KUKA KRL program: EPS_2_25999_MH4A_A_20251114084358.src

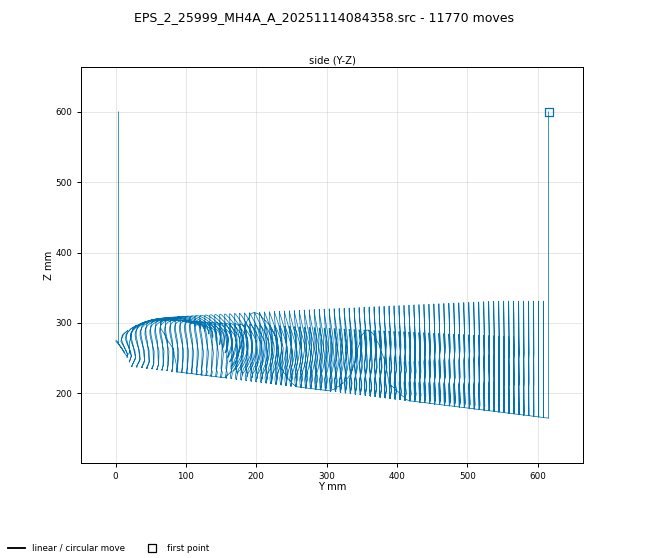
[picture p0: tool path of EPS_2_25999_MH4A_A_20251114084358.src, 11770 of 11772 moves have a stored position in this frame; points joined in program order, loops and branches not executed]
&ACCESS RVP
&REL 4
&COMMENT QRS 19112012
&PARAM EDITMASK = *
DEF PART()
EXT BAS (BAS_COMMAND :IN,REAL :IN )
INT I
BAS (#INITMOV,0 )

;KUKA QRS Post kuka4.cps  Date:22-06-2017 !

File_ID=2914

QRS_PRE_INIT()

;Init var - Until changes are made in qrs_pre_init
Outlet_Square_prg=0
Inlet_1_Square_prg=0
Inlet_2_Square_prg=0
Inlet_3_Square_prg=0
Inlet_4_Square_prg=0
Inlet_5_Square_prg=0

Outlet_1={X 0.000, Y 541.800, Z 256.000, B 0.000, E1 0.000 }
Inlet_1={X 0.000, Y 548.610, Z 213.500, B 0.000, E1 225.000 }
Outlet_1_type=150
Inlet_1_type=135
;QRS#1=Sidecore dimensions
;QRS#2=150-6" PVC SDR 28
;QRS#3=135-5" PVC SDR 28
;QRS#4=
;QRS#5=
;QRS#6=
;QRS#7=
;QRS#8=
;QRS#9=10-06 PSX
;QRS#10=8-11 PSX
;QRS#11=
;QRS#12=
;QRS#13=
;QRS#14=
;QRS#15=
;QRS#16=1220x127x610 2'
;QRS#17=EPS Height
;QRS#18=331
;QRS#19=*
;QRS#20= UPDATED VERSION 22-06-2017
;QRS#21=*
Outlet_Square=070
Inlet_1_Square=070
Inlet_2_Square=0
Inlet_3_Square=0
Inlet_4_Square=0
Inlet_5_Square=0
Mill_Square=1
Outlet_Square_Prg=203
Inlet_1_Square_prg=202

QRS_INIT()

$ADVANCE=5

; T1
PTP {E1 173.61,E2 173.61}
PTP {X 0,Y 615.503,A -85,B 0,C 180,E1 173.61,E2 173.61,E3 0,E4 0,E5 0,E6 0}
QRS_SPEED_INIT()
LIN {X 0,Y 615.503,Z 600,A -85,B 0,C 180,E1 173.61,E2 173.61,E3 0,E4 0,E5 0,E6 0} C_VEL
LIN {X 0,Y 615.503,Z 174.687,A -85,B 0,C 180,E1 173.61,E2 173.61} C_VEL
LIN {X 0,Y 615.503,Z 166.515,A -85,B 0,C 180,E1 173.61,E2 173.61} C_VEL
LIN {X 0,Y 615.489,Z 164.515,A -85,B 0,C 180,E1 173.424,E2 173.424} C_VEL
LIN {X 0,Y 615.497,Z 164.512,A -85,B 0,C 180,E1 170.802,E2 170.802} C_VEL
LIN {X 0,Y 615.481,Z 164.513,A -85,B 0,C 180,E1 168.14,E2 168.14} C_VEL
LIN {X 0,Y 615.485,Z 164.51,A -85,B 0,C 180,E1 165.452,E2 165.452} C_VEL
LIN {X 0,Y 615.477,Z 164.51,A -85,B 0,C 180,E1 162.73,E2 162.73} C_VEL
LIN {X 0,Y 615.462,Z 164.512,A -85,B 0,C 180,E1 159.967,E2 159.967} C_VEL
LIN {X 0,Y 615.491,Z 164.508,A -85,B 0,C 180,E1 157.156,E2 157.156} C_VEL
LIN {X 0,Y 615.498,Z 164.512,A -85,B 0,C 180,E1 154.286,E2 154.286} C_VEL
LIN {X 0,Y 615.493,Z 164.507,A -85,B 0,C 180,E1 151.343,E2 151.343} C_VEL
LIN {X 0,Y 615.477,Z 164.512,A -85,B 0,C 180,E1 148.916,E2 148.916} C_VEL
LIN {X 0,Y 615.487,Z 164.512,A -85,B 0,C 180,E1 146.466,E2 146.466} C_VEL
LIN {X 0,Y 615.49,Z 164.507,A -85,B 0,C 180,E1 143.577,E2 143.577} C_VEL
LIN {X 0,Y 615.463,Z 164.512,A -85,B 0,C 180,E1 140.941,E2 140.941} C_VEL
LIN {X 0,Y 615.467,Z 164.513,A -85,B 0,C 180,E1 138.526,E2 138.526} C_VEL
LIN {X 0,Y 615.494,Z 164.506,A -85,B 0,C 180,E1 135.852,E2 135.852} C_VEL
LIN {X 0,Y 615.463,Z 164.513,A -85,B 0,C 180,E1 133.046,E2 133.046} C_VEL
LIN {X 0,Y 615.46,Z 164.513,A -85,B 0,C 180,E1 130.609,E2 130.609} C_VEL
LIN {X 0,Y 615.488,Z 164.507,A -85,B 0,C 180,E1 128.014,E2 128.014} C_VEL
LIN {X 0,Y 615.474,Z 164.51,A -85,B 0,C 180,E1 125.617,E2 125.617} C_VEL
LIN {X 0,Y 615.468,Z 164.512,A -85,B 0,C 180,E1 123.238,E2 123.238} C_VEL
LIN {X 0,Y 615.485,Z 164.512,A -85,B 0,C 180,E1 120.92,E2 120.92} C_VEL
LIN {X 0,Y 615.496,Z 164.512,A -85,B 0,C 180,E1 118.454,E2 118.454} C_VEL
LIN {X 0,Y 615.468,Z 164.512,A -85,B 0,C 180,E1 115.567,E2 115.567} C_VEL
LIN {X 0,Y 615.476,Z 164.51,A -85,B 0,C 180,E1 112.845,E2 112.845} C_VEL
LIN {X 0,Y 615.481,Z 164.509,A -85,B 0,C 180,E1 110.033,E2 110.033} C_VEL
LIN {X 0,Y 615.471,Z 164.514,A -85,B 0,C 180,E1 107.271,E2 107.271} C_VEL
LIN {X 0,Y 615.494,Z 164.512,A -85,B 0,C 180,E1 104.549,E2 104.549} C_VEL
LIN {X 0,Y 615.486,Z 164.514,A -85,B 0,C 180,E1 101.861,E2 101.861} C_VEL
LIN {X 0,Y 615.494,Z 164.51,A -85,B 0,C 180,E1 99.199,E2 99.199} C_VEL
LIN {X 0,Y 615.477,Z 164.512,A -85,B 0,C 180,E1 96.557,E2 96.557} C_VEL
LIN {X 0,Y 615.472,Z 164.512,A -85,B 0,C 180,E1 93.929,E2 93.929} C_VEL
LIN {X 0,Y 615.488,Z 164.508,A -85,B 0,C 180,E1 91.309,E2 91.309} C_VEL
LIN {X 0,Y 615.474,Z 164.511,A -85,B 0,C 180,E1 88.692,E2 88.692} C_VEL
LIN {X 0,Y 615.464,Z 164.512,A -85,B 0,C 180,E1 86.071,E2 86.071} C_VEL
LIN {X 0,Y 615.487,Z 164.507,A -85,B 0,C 180,E1 83.412,E2 83.412} C_VEL
LIN {X 0,Y 615.475,Z 164.51,A -85,B 0,C 180,E1 80.801,E2 80.801} C_VEL
LIN {X 0,Y 615.464,Z 164.513,A -85,B 0,C 180,E1 78.139,E2 78.139} C_VEL
LIN {X 0,Y 615.476,Z 164.51,A -85,B 0,C 180,E1 76.799,E2 76.799} C_VEL
LIN {X 0,Y 615.481,Z 165.4,A -85,B 0,C 180,E1 76.065,E2 76.065} C_VEL
LIN {X 0,Y 615.489,Z 170.184,A -85,B 0,C 180,E1 73.413,E2 73.413} C_VEL
LIN {X 0,Y 615.478,Z 175.208,A -85,B 0,C 180,E1 70.662,E2 70.662} C_VEL
LIN {X 0,Y 615.453,Z 179.147,A -85,B 0,C 180,E1 68.567,E2 68.567} C_VEL
LIN {X 0,Y 615.485,Z 184.575,A -85,B 0,C 180,E1 65.728,E2 65.728} C_VEL
LIN {X 0,Y 615.43,Z 190.251,A -85,B 0,C 180,E1 62.82,E2 62.82} C_VEL
LIN {X 0,Y 615.497,Z 195.416,A -85,B 0,C 180,E1 60.202,E2 60.202} C_VEL
LIN {X 0,Y 615.471,Z 200.75,A -85,B 0,C 180,E1 57.542,E2 57.542} C_VEL
LIN {X 0,Y 615.477,Z 205.521,A -85,B 0,C 180,E1 55.184,E2 55.184} C_VEL
LIN {X 0,Y 615.486,Z 209.216,A -85,B 0,C 180,E1 53.367,E2 53.367} C_VEL
LIN {X 0,Y 615.484,Z 219.857,A -85,B 0,C 180,E1 53.062,E2 53.062} C_VEL
LIN {X 0,Y 615.474,Z 228.721,A -85,B 0,C 180,E1 52.709,E2 52.709} C_VEL
LIN {X 0,Y 615.482,Z 237.063,A -85,B 0,C 180,E1 52.276,E2 52.276} C_VEL
LIN {X 0,Y 615.489,Z 246.817,A -85,B 0,C 180,E1 51.619,E2 51.619} C_VEL
LIN {X 0,Y 615.496,Z 254.636,A -85,B 0,C 180,E1 50.935,E2 50.935} C_VEL
LIN {X 0,Y 615.499,Z 260.962,A -85,B 0,C 180,E1 50.251,E2 50.251} C_VEL
LIN {X 0,Y 615.495,Z 267.278,A -85,B 0,C 180,E1 49.394,E2 49.394} C_VEL
LIN {X 0,Y 615.495,Z 272.077,A -85,B 0,C 180,E1 48.527,E2 48.527} C_VEL
LIN {X 0,Y 615.496,Z 275.715,A -85,B 0,C 180,E1 47.648,E2 47.648} C_VEL
LIN {X 0,Y 615.495,Z 278.295,A -85,B 0,C 180,E1 46.756,E2 46.756} C_VEL
LIN {X 0,Y 615.492,Z 279.859,A -85,B 0,C 180,E1 45.851,E2 45.851} C_VEL
LIN {X 0,Y 615.498,Z 280.387,A -85,B 0,C 180,E1 44.932,E2 44.932} C_VEL
LIN {X 0,Y 615.493,Z 279.772,A -85,B 0,C 180,E1 43.998,E2 43.998} C_VEL
LIN {X 0,Y 615.493,Z 278.038,A -85,B 0,C 180,E1 43.048,E2 43.048} C_VEL
LIN {X 0,Y 615.499,Z 276.021,A -85,B 0,C 180,E1 42.351,E2 42.351} C_VEL
LIN {X 0,Y 615.493,Z 272.484,A -85,B 0,C 180,E1 41.472,E2 41.472} C_VEL
LIN {X 0,Y 615.494,Z 267.808,A -85,B 0,C 180,E1 40.605,E2 40.605} C_VEL
LIN {X 0,Y 615.497,Z 261.727,A -85,B 0,C 180,E1 39.748,E2 39.748} C_VEL
LIN {X 0,Y 615.496,Z 255.543,A -85,B 0,C 180,E1 39.063,E2 39.063} C_VEL
LIN {X 0,Y 615.491,Z 249.179,A -85,B 0,C 180,E1 38.484,E2 38.484} C_VEL
LIN {X 0,Y 615.445,Z 241.506,A -85,B 0,C 180,E1 37.912,E2 37.912} C_VEL
LIN {X 0,Y 615.443,Z 231.76,A -85,B 0,C 180,E1 37.339,E2 37.339} C_VEL
LIN {X 0,Y 615.473,Z 222.384,A -85,B 0,C 180,E1 36.935,E2 36.935} C_VEL
LIN {X 0,Y 615.497,Z 213.181,A -85,B 0,C 180,E1 36.646,E2 36.646} C_VEL
LIN {X 0,Y 615.488,Z 209.2,A -85,B 0,C 180,E1 36.535,E2 36.535} C_VEL
LIN {X 0,Y 615.462,Z 204.091,A -85,B 0,C 180,E1 34.023,E2 34.023} C_VEL
LIN {X 0,Y 615.48,Z 199.37,A -85,B 0,C 180,E1 31.685,E2 31.685} C_VEL
LIN {X 0,Y 615.482,Z 194.823,A -85,B 0,C 180,E1 29.406,E2 29.406} C_VEL
LIN {X 0,Y 615.474,Z 190.147,A -85,B 0,C 180,E1 27.042,E2 27.042} C_VEL
LIN {X 0,Y 615.486,Z 184.746,A -85,B 0,C 180,E1 24.271,E2 24.271} C_VEL
LIN {X 0,Y 615.446,Z 180.666,A -85,B 0,C 180,E1 22.137,E2 22.137} C_VEL
LIN {X 0,Y 615.428,Z 176.69,A -85,B 0,C 180,E1 20.034,E2 20.034} C_VEL
LIN {X 0,Y 615.495,Z 171.608,A -85,B 0,C 180,E1 17.27,E2 17.27} C_VEL
LIN {X 0,Y 615.465,Z 166.69,A -85,B 0,C 180,E1 14.549,E2 14.549} C_VEL
LIN {X 0,Y 615.496,Z 164.508,A -85,B 0,C 180,E1 13.2,E2 13.2} C_VEL
LIN {X 0,Y 615.474,Z 164.512,A -85,B 0,C 180,E1 10.526,E2 10.526} C_VEL
LIN {X 0,Y 615.487,Z 164.514,A -85,B 0,C 180,E1 7.875,E2 7.875} C_VEL
LIN {X 0,Y 615.491,Z 164.509,A -85,B 0,C 180,E1 5.241,E2 5.241} C_VEL
LIN {X 0,Y 615.47,Z 164.512,A -85,B 0,C 180,E1 2.617,E2 2.617} C_VEL
LIN {X 0,Y 615.482,Z 164.512,A -85,B 0,C 180,E1 -0.001,E2 -0.001} C_VEL
LIN {X 0,Y 615.489,Z 164.512,A -85,B 0,C 180,E1 -2.618,E2 -2.618} C_VEL
LIN {X 0,Y 615.471,Z 164.512,A -85,B 0,C 180,E1 -5.242,E2 -5.242} C_VEL
LIN {X 0,Y 615.474,Z 164.512,A -85,B 0,C 180,E1 -7.876,E2 -7.876} C_VEL
LIN {X 0,Y 615.493,Z 164.514,A -85,B 0,C 180,E1 -10.527,E2 -10.527} C_VEL
LIN {X 0,Y 615.473,Z 164.512,A -85,B 0,C 180,E1 -13.202,E2 -13.202} C_VEL
LIN {X 0,Y 615.489,Z 164.509,A -85,B 0,C 180,E1 -15.906,E2 -15.906} C_VEL
LIN {X 0,Y 615.49,Z 164.512,A -85,B 0,C 180,E1 -18.646,E2 -18.646} C_VEL
LIN {X 0,Y 615.475,Z 164.511,A -85,B 0,C 180,E1 -21.433,E2 -21.433} C_VEL
LIN {X 0,Y 615.489,Z 164.515,A -85,B 0,C 180,E1 -24.272,E2 -24.272} C_VEL
LIN {X 0,Y 615.469,Z 164.513,A -85,B 0,C 180,E1 -27.041,E2 -27.041} C_VEL
LIN {X 0,Y 615.497,Z 164.509,A -85,B 0,C 180,E1 -29.796,E2 -29.796} C_VEL
LIN {X 0,Y 615.482,Z 164.513,A -85,B 0,C 180,E1 -32.458,E2 -32.458} C_VEL
LIN {X 0,Y 615.485,Z 164.512,A -85,B 0,C 180,E1 -34.816,E2 -34.816} C_VEL
LIN {X 0,Y 615.493,Z 164.508,A -85,B 0,C 180,E1 -37.242,E2 -37.242} C_VEL
LIN {X 0,Y 615.483,Z 164.512,A -85,B 0,C 180,E1 -40.088,E2 -40.088} C_VEL
LIN {X 0,Y 615.478,Z 164.513,A -85,B 0,C 180,E1 -42.354,E2 -42.354} C_VEL
LIN {X 0,Y 615.494,Z 164.511,A -85,B 0,C 180,E1 -45.068,E2 -45.068} C_VEL
LIN {X 0,Y 615.472,Z 164.512,A -85,B 0,C 180,E1 -47.922,E2 -47.922} C_VEL
LIN {X 0,Y 615.469,Z 164.513,A -85,B 0,C 180,E1 -50.248,E2 -50.248} C_VEL
LIN {X 0,Y 615.492,Z 164.512,A -85,B 0,C 180,E1 -53.063,E2 -53.063} C_VEL
LIN {X 0,Y 615.472,Z 164.513,A -85,B 0,C 180,E1 -55.977,E2 -55.977} C_VEL
LIN {X 0,Y 615.474,Z 164.512,A -85,B 0,C 180,E1 -58.314,E2 -58.314} C_VEL
LIN {X 0,Y 615.478,Z 164.615,A -85,B 0,C 180,E1 -59.46,E2 -59.46} C_VEL
LIN {X 0,Y 615.479,Z 174.178,A -85,B 0,C 180,E1 -62.085,E2 -62.085} C_VEL
LIN {X 0,Y 615.463,Z 185.21,A -85,B 0,C 180,E1 -65.007,E2 -65.007} C_VEL
LIN {X 0,Y 615.452,Z 193.485,A -85,B 0,C 180,E1 -67.154,E2 -67.154} C_VEL
LIN {X 0,Y 615.469,Z 203.484,A -85,B 0,C 180,E1 -69.709,E2 -69.709} C_VEL
LIN {X 0,Y 615.495,Z 214.135,A -85,B 0,C 180,E1 -72.387,E2 -72.387} C_VEL
LIN {X 0,Y 615.473,Z 225.145,A -85,B 0,C 180,E1 -75.112,E2 -75.112} C_VEL
LIN {X 0,Y 615.479,Z 236.141,A -85,B 0,C 180,E1 -77.805,E2 -77.805} C_VEL
LIN {X 0,Y 615.489,Z 247.136,A -85,B 0,C 180,E1 -80.47,E2 -80.47} C_VEL
LIN {X 0,Y 615.485,Z 248.505,A -85,B 0,C 180,E1 -80.801,E2 -80.801} C_VEL
LIN {X 0,Y 615.495,Z 260.895,A -85,B 0,C 180,E1 -81.091,E2 -81.091} C_VEL
LIN {X 0,Y 615.471,Z 271.229,A -85,B 0,C 180,E1 -81.463,E2 -81.463} C_VEL
LIN {X 0,Y 615.474,Z 279.916,A -85,B 0,C 180,E1 -81.877,E2 -81.877} C_VEL
LIN {X 0,Y 615.492,Z 288.199,A -85,B 0,C 180,E1 -82.372,E2 -82.372} C_VEL
LIN {X 0,Y 615.499,Z 295.935,A -85,B 0,C 180,E1 -82.942,E2 -82.942} C_VEL
LIN {X 0,Y 615.498,Z 301.647,A -85,B 0,C 180,E1 -83.444,E2 -83.444} C_VEL
LIN {X 0,Y 615.5,Z 307.922,A -85,B 0,C 180,E1 -84.102,E2 -84.102} C_VEL
LIN {X 0,Y 615.495,Z 313.136,A -85,B 0,C 180,E1 -84.759,E2 -84.759} C_VEL
LIN {X 0,Y 615.495,Z 317.483,A -85,B 0,C 180,E1 -85.416,E2 -85.416} C_VEL
LIN {X 0,Y 615.491,Z 322.604,A -85,B 0,C 180,E1 -86.399,E2 -86.399} C_VEL
LIN {X 0,Y 615.488,Z 325.221,A -85,B 0,C 180,E1 -87.055,E2 -87.055} C_VEL
LIN {X 0,Y 615.499,Z 328.085,A -85,B 0,C 180,E1 -88.037,E2 -88.037} C_VEL
LIN {X 0,Y 615.493,Z 329.33,A -85,B 0,C 180,E1 -88.692,E2 -88.692} C_VEL
LIN {X 0,Y 615.491,Z 330.104,A -85,B 0,C 180,E1 -89.346,E2 -89.346} C_VEL
LIN {X 0,Y 615.491,Z 330.389,A -85,B 0,C 180,E1 -90,E2 -90} C_VEL
LIN {X 0,Y 615.491,Z 330.104,A -85,B 0,C 180,E1 -90.654,E2 -90.654} C_VEL
LIN {X 0,Y 615.493,Z 329.33,A -85,B 0,C 180,E1 -91.309,E2 -91.309} C_VEL
LIN {X 0,Y 615.499,Z 328.085,A -85,B 0,C 180,E1 -91.963,E2 -91.963} C_VEL
LIN {X 0,Y 615.488,Z 325.22,A -85,B 0,C 180,E1 -92.945,E2 -92.945} C_VEL
LIN {X 0,Y 615.491,Z 322.603,A -85,B 0,C 180,E1 -93.601,E2 -93.601} C_VEL
LIN {X 0,Y 615.495,Z 317.482,A -85,B 0,C 180,E1 -94.585,E2 -94.585} C_VEL
LIN {X 0,Y 615.495,Z 311.967,A -85,B 0,C 180,E1 -95.406,E2 -95.406} C_VEL
LIN {X 0,Y 615.498,Z 305.016,A -85,B 0,C 180,E1 -96.228,E2 -96.228} C_VEL
LIN {X 0,Y 615.498,Z 297.858,A -85,B 0,C 180,E1 -96.901,E2 -96.901} C_VEL
LIN {X 0,Y 615.489,Z 290.619,A -85,B 0,C 180,E1 -97.463,E2 -97.463} C_VEL
LIN {X 0,Y 615.482,Z 282.869,A -85,B 0,C 180,E1 -97.958,E2 -97.958} C_VEL
LIN {X 0,Y 615.468,Z 274.917,A -85,B 0,C 180,E1 -98.372,E2 -98.372} C_VEL
LIN {X 0,Y 615.481,Z 265.754,A -85,B 0,C 180,E1 -98.744,E2 -98.744} C_VEL
LIN {X 0,Y 615.493,Z 257.686,A -85,B 0,C 180,E1 -98.992,E2 -98.992} C_VEL
LIN {X 0,Y 615.485,Z 248.504,A -85,B 0,C 180,E1 -99.199,E2 -99.199} C_VEL
LIN {X 0,Y 615.487,Z 237.518,A -85,B 0,C 180,E1 -101.861,E2 -101.861} C_VEL
LIN {X 0,Y 615.492,Z 226.514,A -85,B 0,C 180,E1 -104.549,E2 -104.549} C_VEL
LIN {X 0,Y 615.479,Z 215.517,A -85,B 0,C 180,E1 -107.271,E2 -107.271} C_VEL
LIN {X 0,Y 615.487,Z 204.497,A -85,B 0,C 180,E1 -110.033,E2 -110.033} C_VEL
LIN {X 0,Y 615.452,Z 195.46,A -85,B 0,C 180,E1 -112.338,E2 -112.338} C_VEL
LIN {X 0,Y 615.441,Z 186.593,A -85,B 0,C 180,E1 -114.634,E2 -114.634} C_VEL
LIN {X 0,Y 615.479,Z 176.933,A -85,B 0,C 180,E1 -117.178,E2 -117.178} C_VEL
LIN {X 0,Y 615.48,Z 167.272,A -85,B 0,C 180,E1 -119.793,E2 -119.793} C_VEL
LIN {X 0,Y 615.478,Z 164.51,A -85,B 0,C 180,E1 -120.587,E2 -120.587} C_VEL
LIN {X 0,Y 615.478,Z 164.509,A -85,B 0,C 180,E1 -123.533,E2 -123.533} C_VEL
LIN {X 0,Y 615.477,Z 164.514,A -85,B 0,C 180,E1 -126.426,E2 -126.426} C_VEL
LIN {X 0,Y 615.499,Z 164.511,A -85,B 0,C 180,E1 -129.063,E2 -129.063} C_VEL
LIN {X 0,Y 615.484,Z 164.512,A -85,B 0,C 180,E1 -131.474,E2 -131.474} C_VEL
LIN {X 0,Y 615.491,Z 164.513,A -85,B 0,C 180,E1 -134.15,E2 -134.15} C_VEL
LIN {X 0,Y 615.481,Z 164.513,A -85,B 0,C 180,E1 -136.954,E2 -136.954} C_VEL
LIN {X 0,Y 615.483,Z 164.515,A -85,B 0,C 180,E1 -139.393,E2 -139.393} C_VEL
LIN {X 0,Y 615.488,Z 164.513,A -85,B 0,C 180,E1 -141.988,E2 -141.988} C_VEL
LIN {X 0,Y 615.491,Z 164.513,A -85,B 0,C 180,E1 -144.384,E2 -144.384} C_VEL
LIN {X 0,Y 615.492,Z 164.509,A -85,B 0,C 180,E1 -146.764,E2 -146.764} C_VEL
LIN {X 0,Y 615.469,Z 164.511,A -85,B 0,C 180,E1 -149.079,E2 -149.079} C_VEL
LIN {X 0,Y 615.463,Z 164.512,A -85,B 0,C 180,E1 -151.555,E2 -151.555} C_VEL
LIN {X 0,Y 615.495,Z 164.508,A -85,B 0,C 180,E1 -154.43,E2 -154.43} C_VEL
LIN {X 0,Y 615.488,Z 164.514,A -85,B 0,C 180,E1 -157.155,E2 -157.155} C_VEL
LIN {X 0,Y 615.493,Z 164.51,A -85,B 0,C 180,E1 -159.967,E2 -159.967} C_VEL
LIN {X 0,Y 615.467,Z 164.512,A -85,B 0,C 180,E1 -162.729,E2 -162.729} C_VEL
LIN {X 0,Y 615.475,Z 164.51,A -85,B 0,C 180,E1 -165.45,E2 -165.45} C_VEL
LIN {X 0,Y 615.484,Z 164.508,A -85,B 0,C 180,E1 -168.139,E2 -168.139} C_VEL
LIN {X 0,Y 615.465,Z 164.512,A -85,B 0,C 180,E1 -170.8,E2 -170.8} C_VEL
LIN {X 0,Y 615.481,Z 164.51,A -85,B 0,C 180,E1 -173.443,E2 -173.443} C_VEL
LIN {X 0,Y 615.488,Z 164.509,A -85,B 0,C 180,E1 -176.071,E2 -176.071} C_VEL
LIN {X 0,Y 615.474,Z 164.513,A -85,B 0,C 180,E1 -178.691,E2 -178.691} C_VEL
LIN {X 0,Y 615.485,Z 164.512,A -85,B 0,C 180,E1 -181.308,E2 -181.308} C_VEL
LIN {X 0,Y 615.49,Z 164.512,A -85,B 0,C 180,E1 -183.928,E2 -183.928} C_VEL
LIN {X 0,Y 615.489,Z 164.515,A -85,B 0,C 180,E1 -186.576,E2 -186.576} C_VEL
LIN {X 0,Y 614.816,Z 164.654,A -85,B 0,C 180,E1 -187.122,E2 -187.122} C_VEL
LIN {X 0,Y 611.989,Z 165.069,A -85,B 0,C 180,E1 -188.008,E2 -188.008} C_VEL
LIN {X 0,Y 609.598,Z 165.379,A -85,B 0,C 180,E1 -188.72,E2 -188.72} C_VEL
LIN {X 0,Y 608.555,Z 165.497,A -85,B 0,C 180,E1 -189.27,E2 -189.27} C_VEL
LIN {X 0,Y 608.461,Z 165.506,A -85,B 0,C 180,E1 -189.456,E2 -189.456} C_VEL
LIN {X 0,Y 608.455,Z 165.507,A -85,B 0,C 180,E1 -191.999,E2 -191.999} C_VEL
LIN {X 0,Y 608.477,Z 165.504,A -85,B 0,C 180,E1 -194.72,E2 -194.72} C_VEL
LIN {X 0,Y 608.448,Z 165.507,A -85,B 0,C 180,E1 -197.476,E2 -197.476} C_VEL
LIN {X 0,Y 608.451,Z 165.507,A -85,B 0,C 180,E1 -200.274,E2 -200.274} C_VEL
LIN {X 0,Y 608.46,Z 165.505,A -85,B 0,C 180,E1 -202.475,E2 -202.475} C_VEL
LIN {X 0,Y 608.451,Z 165.507,A -85,B 0,C 180,E1 -205.3,E2 -205.3} C_VEL
LIN {X 0,Y 608.442,Z 165.508,A -85,B 0,C 180,E1 -207.517,E2 -207.517} C_VEL
LIN {X 0,Y 608.46,Z 165.506,A -85,B 0,C 180,E1 -209.97,E2 -209.97} C_VEL
LIN {X 0,Y 608.462,Z 165.505,A -85,B 0,C 180,E1 -212.878,E2 -212.878} C_VEL
LIN {X 0,Y 608.434,Z 165.508,A -85,B 0,C 180,E1 -215.277,E2 -215.277} C_VEL
LIN {X 0,Y 608.46,Z 165.505,A -85,B 0,C 180,E1 -217.746,E2 -217.746} C_VEL
LIN {X 0,Y 608.479,Z 165.503,A -85,B 0,C 180,E1 -220.332,E2 -220.332} C_VEL
LIN {X 0,Y 608.459,Z 165.507,A -85,B 0,C 180,E1 -223.307,E2 -223.307} C_VEL
LIN {X 0,Y 608.462,Z 165.509,A -85,B 0,C 180,E1 -226.13,E2 -226.13} C_VEL
LIN {X 0,Y 608.449,Z 165.51,A -85,B 0,C 180,E1 -228.823,E2 -228.823} C_VEL
LIN {X 0,Y 608.467,Z 165.505,A -85,B 0,C 180,E1 -231.758,E2 -231.758} C_VEL
LIN {X 0,Y 608.439,Z 165.509,A -85,B 0,C 180,E1 -234.722,E2 -234.722} C_VEL
LIN {X 0,Y 608.461,Z 165.508,A -85,B 0,C 180,E1 -237.476,E2 -237.476} C_VEL
LIN {X 0,Y 608.481,Z 165.507,A -85,B 0,C 180,E1 -240.221,E2 -240.221} C_VEL
LIN {X 0,Y 608.478,Z 165.508,A -85,B 0,C 180,E1 -242.791,E2 -242.791} C_VEL
LIN {X 0,Y 608.477,Z 165.503,A -85,B 0,C 180,E1 -245.845,E2 -245.845} C_VEL
LIN {X 0,Y 608.458,Z 165.506,A -85,B 0,C 180,E1 -248.308,E2 -248.308} C_VEL
LIN {X 0,Y 608.452,Z 165.506,A -85,B 0,C 180,E1 -251.13,E2 -251.13} C_VEL
LIN {X 0,Y 608.462,Z 165.506,A -85,B 0,C 180,E1 -253.906,E2 -253.906} C_VEL
LIN {X 0,Y 608.463,Z 165.507,A -85,B 0,C 180,E1 -256.643,E2 -256.643} C_VEL
LIN {X 0,Y 608.461,Z 165.51,A -85,B 0,C 180,E1 -259.35,E2 -259.35} C_VEL
LIN {X 0,Y 608.472,Z 165.507,A -85,B 0,C 180,E1 -262.033,E2 -262.033} C_VEL
LIN {X 0,Y 608.467,Z 165.507,A -85,B 0,C 180,E1 -264.698,E2 -264.698} C_VEL
LIN {X 0,Y 608.465,Z 165.506,A -85,B 0,C 180,E1 -267.352,E2 -267.352} C_VEL
LIN {X 0,Y 608.455,Z 165.507,A -85,B 0,C 180,E1 -270,E2 -270} C_VEL
LIN {X 0,Y 608.477,Z 165.503,A -85,B 0,C 180,E1 -272.648,E2 -272.648} C_VEL
LIN {X 0,Y 608.456,Z 165.506,A -85,B 0,C 180,E1 -275.302,E2 -275.302} C_VEL
LIN {X 0,Y 608.46,Z 165.505,A -85,B 0,C 180,E1 -277.967,E2 -277.967} C_VEL
LIN {X 0,Y 608.465,Z 165.505,A -85,B 0,C 180,E1 -280.65,E2 -280.65} C_VEL
LIN {X 0,Y 608.421,Z 165.512,A -85,B 0,C 180,E1 -283.357,E2 -283.357} C_VEL
LIN {X 0,Y 608.449,Z 168.953,A -85,B 0,C 180,E1 -285.406,E2 -285.406} C_VEL
LIN {X 0,Y 608.451,Z 173.943,A -85,B 0,C 180,E1 -288.172,E2 -288.172} C_VEL
LIN {X 0,Y 608.428,Z 179.12,A -85,B 0,C 180,E1 -290.982,E2 -290.982} C_VEL
LIN {X 0,Y 608.409,Z 183.175,A -85,B 0,C 180,E1 -293.126,E2 -293.126} C_VEL
LIN {X 0,Y 608.38,Z 188.138,A -85,B 0,C 180,E1 -295.705,E2 -295.705} C_VEL
LIN {X 0,Y 608.396,Z 193.813,A -85,B 0,C 180,E1 -298.609,E2 -298.609} C_VEL
LIN {X 0,Y 608.411,Z 197.653,A -85,B 0,C 180,E1 -300.548,E2 -300.548} C_VEL
LIN {X 0,Y 608.402,Z 202.321,A -85,B 0,C 180,E1 -302.883,E2 -302.883} C_VEL
LIN {X 0,Y 608.399,Z 207.157,A -85,B 0,C 180,E1 -305.281,E2 -305.281} C_VEL
LIN {X 0,Y 608.416,Z 209.693,A -85,B 0,C 180,E1 -306.531,E2 -306.531} C_VEL
LIN {X 0,Y 608.487,Z 220.755,A -85,B 0,C 180,E1 -306.861,E2 -306.861} C_VEL
LIN {X 0,Y 608.46,Z 230.422,A -85,B 0,C 180,E1 -307.26,E2 -307.26} C_VEL
LIN {X 0,Y 608.461,Z 241.137,A -85,B 0,C 180,E1 -307.87,E2 -307.87} C_VEL
LIN {X 0,Y 608.46,Z 249.454,A -85,B 0,C 180,E1 -308.487,E2 -308.487} C_VEL
LIN {X 0,Y 608.445,Z 256.717,A -85,B 0,C 180,E1 -309.156,E2 -309.156} C_VEL
LIN {X 0,Y 608.467,Z 262.956,A -85,B 0,C 180,E1 -309.87,E2 -309.87} C_VEL
LIN {X 0,Y 608.436,Z 268.87,A -85,B 0,C 180,E1 -310.74,E2 -310.74} C_VEL
LIN {X 0,Y 608.431,Z 272.203,A -85,B 0,C 180,E1 -311.34,E2 -311.34} C_VEL
LIN {X 0,Y 608.437,Z 276.332,A -85,B 0,C 180,E1 -312.333,E2 -312.333} C_VEL
LIN {X 0,Y 608.431,Z 279.091,A -85,B 0,C 180,E1 -313.306,E2 -313.306} C_VEL
LIN {X 0,Y 608.42,Z 280.624,A -85,B 0,C 180,E1 -314.262,E2 -314.262} C_VEL
LIN {X 0,Y 608.418,Z 280.951,A -85,B 0,C 180,E1 -315.202,E2 -315.202} C_VEL
LIN {X 0,Y 608.428,Z 280.216,A -85,B 0,C 180,E1 -316.128,E2 -316.128} C_VEL
LIN {X 0,Y 608.434,Z 278.473,A -85,B 0,C 180,E1 -317.04,E2 -317.04} C_VEL
LIN {X 0,Y 608.427,Z 275.709,A -85,B 0,C 180,E1 -317.937,E2 -317.937} C_VEL
LIN {X 0,Y 608.438,Z 270.645,A -85,B 0,C 180,E1 -319.043,E2 -319.043} C_VEL
LIN {X 0,Y 608.443,Z 265.159,A -85,B 0,C 180,E1 -319.914,E2 -319.914} C_VEL
LIN {X 0,Y 608.455,Z 258.851,A -85,B 0,C 180,E1 -320.704,E2 -320.704} C_VEL
LIN {X 0,Y 608.459,Z 250.521,A -85,B 0,C 180,E1 -321.515,E2 -321.515} C_VEL
LIN {X 0,Y 608.422,Z 242.468,A -85,B 0,C 180,E1 -322.13,E2 -322.13} C_VEL
LIN {X 0,Y 608.432,Z 233.724,A -85,B 0,C 180,E1 -322.661,E2 -322.661} C_VEL
LIN {X 0,Y 608.481,Z 223.325,A -85,B 0,C 180,E1 -323.14,E2 -323.14} C_VEL
LIN {X 0,Y 608.485,Z 212.694,A -85,B 0,C 180,E1 -323.475,E2 -323.475} C_VEL
LIN {X 0,Y 608.426,Z 209.688,A -85,B 0,C 180,E1 -323.561,E2 -323.561} C_VEL
LIN {X 0,Y 608.404,Z 204.092,A -85,B 0,C 180,E1 -326.327,E2 -326.327} C_VEL
LIN {X 0,Y 608.415,Z 199.256,A -85,B 0,C 180,E1 -328.737,E2 -328.737} C_VEL
LIN {X 0,Y 608.428,Z 193.995,A -85,B 0,C 180,E1 -331.388,E2 -331.388} C_VEL
LIN {X 0,Y 608.406,Z 188.316,A -85,B 0,C 180,E1 -334.292,E2 -334.292} C_VEL
LIN {X 0,Y 608.421,Z 183.344,A -85,B 0,C 180,E1 -336.876,E2 -336.876} C_VEL
LIN {X 0,Y 608.39,Z 177.969,A -85,B 0,C 180,E1 -339.724,E2 -339.724} C_VEL
LIN {X 0,Y 608.453,Z 172.859,A -85,B 0,C 180,E1 -342.524,E2 -342.524} C_VEL
LIN {X 0,Y 608.432,Z 167.917,A -85,B 0,C 180,E1 -345.279,E2 -345.279} C_VEL
LIN {X 0,Y 608.431,Z 165.512,A -85,B 0,C 180,E1 -346.644,E2 -346.644} C_VEL
LIN {X 0,Y 608.455,Z 165.507,A -85,B 0,C 180,E1 -349.351,E2 -349.351} C_VEL
LIN {X 0,Y 608.476,Z 165.506,A -85,B 0,C 180,E1 -352.034,E2 -352.034} C_VEL
LIN {X 0,Y 608.469,Z 165.507,A -85,B 0,C 180,E1 -354.699,E2 -354.699} C_VEL
LIN {X 0,Y 608.463,Z 165.506,A -85,B 0,C 180,E1 -357.352,E2 -357.352} C_VEL
LIN {X 0,Y 608.474,Z 165.506,A -85,B 0,C 180,E1 -360.001,E2 -360.001} C_VEL
LIN {X 0,Y 608.479,Z 165.506,A -85,B 0,C 180,E1 -362.649,E2 -362.649} C_VEL
LIN {X 0,Y 608.454,Z 165.507,A -85,B 0,C 180,E1 -365.302,E2 -365.302} C_VEL
LIN {X 0,Y 608.469,Z 165.506,A -85,B 0,C 180,E1 -367.968,E2 -367.968} C_VEL
LIN {X 0,Y 608.464,Z 165.508,A -85,B 0,C 180,E1 -370.65,E2 -370.65} C_VEL
LIN {X 0,Y 608.456,Z 165.507,A -85,B 0,C 180,E1 -373.357,E2 -373.357} C_VEL
LIN {X 0,Y 608.462,Z 165.508,A -85,B 0,C 180,E1 -376.094,E2 -376.094} C_VEL
LIN {X 0,Y 608.456,Z 165.507,A -85,B 0,C 180,E1 -378.87,E2 -378.87} C_VEL
LIN {X 0,Y 608.462,Z 165.507,A -85,B 0,C 180,E1 -381.692,E2 -381.692} C_VEL
LIN {X 0,Y 608.45,Z 165.508,A -85,B 0,C 180,E1 -384.572,E2 -384.572} C_VEL
LIN {X 0,Y 608.465,Z 165.506,A -85,B 0,C 180,E1 -387.205,E2 -387.205} C_VEL
LIN {X 0,Y 608.474,Z 165.508,A -85,B 0,C 180,E1 -389.972,E2 -389.972} C_VEL
LIN {X 0,Y 608.455,Z 165.507,A -85,B 0,C 180,E1 -392.88,E2 -392.88} C_VEL
LIN {X 0,Y 608.449,Z 165.508,A -85,B 0,C 180,E1 -395.278,E2 -395.278} C_VEL
LIN {X 0,Y 608.473,Z 165.506,A -85,B 0,C 180,E1 -397.746,E2 -397.746} C_VEL
LIN {X 0,Y 608.447,Z 165.512,A -85,B 0,C 180,E1 -400.328,E2 -400.328} C_VEL
LIN {X 0,Y 608.479,Z 165.504,A -85,B 0,C 180,E1 -403.31,E2 -403.31} C_VEL
LIN {X 0,Y 608.469,Z 165.508,A -85,B 0,C 180,E1 -406.131,E2 -406.131} C_VEL
LIN {X 0,Y 608.457,Z 165.507,A -85,B 0,C 180,E1 -408.824,E2 -408.824} C_VEL
LIN {X 0,Y 608.469,Z 165.509,A -85,B 0,C 180,E1 -411.76,E2 -411.76} C_VEL
LIN {X 0,Y 608.449,Z 165.51,A -85,B 0,C 180,E1 -413.954,E2 -413.954} C_VEL
LIN {X 0,Y 608.465,Z 165.509,A -85,B 0,C 180,E1 -416.329,E2 -416.329} C_VEL
LIN {X 0,Y 608.471,Z 165.506,A -85,B 0,C 180,E1 -419.287,E2 -419.287} C_VEL
LIN {X 0,Y 608.51,Z 174.243,A -85,B 0,C 180,E1 -421.736,E2 -421.736} C_VEL
LIN {X 0,Y 608.486,Z 183.676,A -85,B 0,C 180,E1 -424.276,E2 -424.276} C_VEL
LIN {X 0,Y 608.453,Z 193.573,A -85,B 0,C 180,E1 -426.876,E2 -426.876} C_VEL
LIN {X 0,Y 608.443,Z 203.078,A -85,B 0,C 180,E1 -429.327,E2 -429.327} C_VEL
LIN {X 0,Y 608.483,Z 214.314,A -85,B 0,C 180,E1 -432.177,E2 -432.177} C_VEL
LIN {X 0,Y 608.428,Z 225.376,A -85,B 0,C 180,E1 -434.936,E2 -434.936} C_VEL
LIN {X 0,Y 608.457,Z 235.056,A -85,B 0,C 180,E1 -437.323,E2 -437.323} C_VEL
LIN {X 0,Y 608.439,Z 246.118,A -85,B 0,C 180,E1 -440.022,E2 -440.022} C_VEL
LIN {X 0,Y 608.427,Z 248.883,A -85,B 0,C 180,E1 -440.694,E2 -440.694} C_VEL
LIN {X 0,Y 608.502,Z 261.237,A -85,B 0,C 180,E1 -440.988,E2 -440.988} C_VEL
LIN {X 0,Y 608.471,Z 271.536,A -85,B 0,C 180,E1 -441.364,E2 -441.364} C_VEL
LIN {X 0,Y 608.455,Z 280.234,A -85,B 0,C 180,E1 -441.782,E2 -441.782} C_VEL
LIN {X 0,Y 608.47,Z 288.543,A -85,B 0,C 180,E1 -442.284,E2 -442.284} C_VEL
LIN {X 0,Y 608.464,Z 296.402,A -85,B 0,C 180,E1 -442.867,E2 -442.867} C_VEL
LIN {X 0,Y 608.466,Z 303.358,A -85,B 0,C 180,E1 -443.496,E2 -443.496} C_VEL
LIN {X 0,Y 608.47,Z 311.192,A -85,B 0,C 180,E1 -444.366,E2 -444.366} C_VEL
LIN {X 0,Y 608.448,Z 317.028,A -85,B 0,C 180,E1 -445.196,E2 -445.196} C_VEL
LIN {X 0,Y 608.434,Z 321.631,A -85,B 0,C 180,E1 -446.026,E2 -446.026} C_VEL
LIN {X 0,Y 608.424,Z 324.622,A -85,B 0,C 180,E1 -446.689,E2 -446.689} C_VEL
LIN {X 0,Y 608.423,Z 326.931,A -85,B 0,C 180,E1 -447.352,E2 -447.352} C_VEL
LIN {X 0,Y 608.444,Z 328.678,A -85,B 0,C 180,E1 -448.014,E2 -448.014} C_VEL
LIN {X 0,Y 608.445,Z 329.934,A -85,B 0,C 180,E1 -448.676,E2 -448.676} C_VEL
LIN {X 0,Y 608.434,Z 330.714,A -85,B 0,C 180,E1 -449.338,E2 -449.338} C_VEL
LIN {X 0,Y 608.431,Z 331,A -85,B 0,C 180,E1 -450,E2 -450} C_VEL
LIN {X 0,Y 608.434,Z 330.714,A -85,B 0,C 180,E1 -450.662,E2 -450.662} C_VEL
LIN {X 0,Y 608.445,Z 329.933,A -85,B 0,C 180,E1 -451.324,E2 -451.324} C_VEL
LIN {X 0,Y 608.444,Z 328.678,A -85,B 0,C 180,E1 -451.986,E2 -451.986} C_VEL
LIN {X 0,Y 608.444,Z 325.785,A -85,B 0,C 180,E1 -452.98,E2 -452.98} C_VEL
LIN {X 0,Y 608.445,Z 323.145,A -85,B 0,C 180,E1 -453.643,E2 -453.643} C_VEL
LIN {X 0,Y 608.431,Z 317.984,A -85,B 0,C 180,E1 -454.638,E2 -454.638} C_VEL
LIN {X 0,Y 608.46,Z 312.429,A -85,B 0,C 180,E1 -455.468,E2 -455.468} C_VEL
LIN {X 0,Y 608.455,Z 304.672,A -85,B 0,C 180,E1 -456.375,E2 -456.375} C_VEL
LIN {X 0,Y 608.484,Z 297.413,A -85,B 0,C 180,E1 -457.049,E2 -457.049} C_VEL
LIN {X 0,Y 608.471,Z 289.758,A -85,B 0,C 180,E1 -457.633,E2 -457.633} C_VEL
LIN {X 0,Y 608.476,Z 281.716,A -85,B 0,C 180,E1 -458.134,E2 -458.134} C_VEL
LIN {X 0,Y 608.478,Z 273.385,A -85,B 0,C 180,E1 -458.552,E2 -458.552} C_VEL
LIN {X 0,Y 608.485,Z 264.883,A -85,B 0,C 180,E1 -458.887,E2 -458.887} C_VEL
LIN {X 0,Y 608.506,Z 255.578,A -85,B 0,C 180,E1 -459.159,E2 -459.159} C_VEL
LIN {X 0,Y 608.426,Z 248.882,A -85,B 0,C 180,E1 -459.307,E2 -459.307} C_VEL
LIN {X 0,Y 608.43,Z 237.82,A -85,B 0,C 180,E1 -462.001,E2 -462.001} C_VEL
LIN {X 0,Y 608.444,Z 226.758,A -85,B 0,C 180,E1 -464.721,E2 -464.721} C_VEL
LIN {X 0,Y 608.462,Z 215.696,A -85,B 0,C 180,E1 -467.476,E2 -467.476} C_VEL
LIN {X 0,Y 608.453,Z 204.634,A -85,B 0,C 180,E1 -470.275,E2 -470.275} C_VEL
LIN {X 0,Y 608.431,Z 194.956,A -85,B 0,C 180,E1 -472.765,E2 -472.765} C_VEL
LIN {X 0,Y 608.483,Z 185.275,A -85,B 0,C 180,E1 -475.3,E2 -475.3} C_VEL
LIN {X 0,Y 608.496,Z 174.218,A -85,B 0,C 180,E1 -478.265,E2 -478.265} C_VEL
LIN {X 0,Y 608.451,Z 165.507,A -85,B 0,C 180,E1 -480.69,E2 -480.69} C_VEL
LIN {X 0,Y 608.453,Z 165.509,A -85,B 0,C 180,E1 -482.88,E2 -482.88} C_VEL
LIN {X 0,Y 608.433,Z 165.513,A -85,B 0,C 180,E1 -485.279,E2 -485.279} C_VEL
LIN {X 0,Y 608.468,Z 165.508,A -85,B 0,C 180,E1 -487.747,E2 -487.747} C_VEL
LIN {X 0,Y 608.447,Z 165.511,A -85,B 0,C 180,E1 -490.328,E2 -490.328} C_VEL
LIN {X 0,Y 608.462,Z 165.506,A -85,B 0,C 180,E1 -493.308,E2 -493.308} C_VEL
LIN {X 0,Y 608.459,Z 165.506,A -85,B 0,C 180,E1 -496.129,E2 -496.129} C_VEL
LIN {X 0,Y 608.459,Z 165.506,A -85,B 0,C 180,E1 -498.824,E2 -498.824} C_VEL
LIN {X 0,Y 608.467,Z 165.507,A -85,B 0,C 180,E1 -501.76,E2 -501.76} C_VEL
LIN {X 0,Y 608.444,Z 165.508,A -85,B 0,C 180,E1 -503.955,E2 -503.955} C_VEL
LIN {X 0,Y 608.471,Z 165.504,A -85,B 0,C 180,E1 -506.329,E2 -506.329} C_VEL
LIN {X 0,Y 608.445,Z 165.508,A -85,B 0,C 180,E1 -508.733,E2 -508.733} C_VEL
LIN {X 0,Y 608.455,Z 165.506,A -85,B 0,C 180,E1 -511.384,E2 -511.384} C_VEL
LIN {X 0,Y 608.481,Z 165.503,A -85,B 0,C 180,E1 -514.278,E2 -514.278} C_VEL
LIN {X 0,Y 608.45,Z 165.508,A -85,B 0,C 180,E1 -516.876,E2 -516.876} C_VEL
LIN {X 0,Y 608.456,Z 165.506,A -85,B 0,C 180,E1 -519.325,E2 -519.325} C_VEL
LIN {X 0,Y 608.453,Z 165.506,A -85,B 0,C 180,E1 -521.828,E2 -521.828} C_VEL
LIN {X 0,Y 608.476,Z 165.505,A -85,B 0,C 180,E1 -524.594,E2 -524.594} C_VEL
LIN {X 0,Y 608.475,Z 165.507,A -85,B 0,C 180,E1 -527.323,E2 -527.323} C_VEL
LIN {X 0,Y 608.452,Z 165.51,A -85,B 0,C 180,E1 -530.022,E2 -530.022} C_VEL
LIN {X 0,Y 608.446,Z 165.51,A -85,B 0,C 180,E1 -532.7,E2 -532.7} C_VEL
LIN {X 0,Y 608.46,Z 165.507,A -85,B 0,C 180,E1 -535.362,E2 -535.362} C_VEL
LIN {X 0,Y 608.438,Z 165.509,A -85,B 0,C 180,E1 -538.014,E2 -538.014} C_VEL
LIN {X 0,Y 608.463,Z 165.505,A -85,B 0,C 180,E1 -540.661,E2 -540.661} C_VEL
LIN {X 0,Y 608.482,Z 165.503,A -85,B 0,C 180,E1 -543.31,E2 -543.31} C_VEL
LIN {X 0,Y 608.443,Z 165.507,A -85,B 0,C 180,E1 -545.966,E2 -545.966} C_VEL
LIN {X 0,Y 608.44,Z 165.508,A -85,B 0,C 180,E1 -548.636,E2 -548.636} C_VEL
LIN {X 0,Y 608.461,Z 165.506,A -85,B 0,C 180,E1 -549.456,E2 -549.456} C_VEL
LIN {X 0,Y 607.771,Z 165.593,A -85,B 0,C 180,E1 -550.009,E2 -550.009} C_VEL
LIN {X 0,Y 604.914,Z 165.947,A -85,B 0,C 180,E1 -550.906,E2 -550.906} C_VEL
LIN {X 0,Y 602.515,Z 166.25,A -85,B 0,C 180,E1 -551.627,E2 -551.627} C_VEL
LIN {X 0,Y 601.486,Z 166.375,A -85,B 0,C 180,E1 -552.184,E2 -552.184} C_VEL
LIN {X 0,Y 601.402,Z 166.385,A -85,B 0,C 180,E1 -552.372,E2 -552.372} C_VEL
LIN {X 0,Y 601.432,Z 166.381,A -85,B 0,C 180,E1 -554.896,E2 -554.896} C_VEL
LIN {X 0,Y 601.394,Z 166.386,A -85,B 0,C 180,E1 -557.688,E2 -557.688} C_VEL
LIN {X 0,Y 601.428,Z 166.384,A -85,B 0,C 180,E1 -560.521,E2 -560.521} C_VEL
LIN {X 0,Y 601.391,Z 166.388,A -85,B 0,C 180,E1 -563.411,E2 -563.411} C_VEL
LIN {X 0,Y 601.417,Z 166.386,A -85,B 0,C 180,E1 -565.867,E2 -565.867} C_VEL
LIN {X 0,Y 601.439,Z 166.381,A -85,B 0,C 180,E1 -568.625,E2 -568.625} C_VEL
LIN {X 0,Y 601.416,Z 166.383,A -85,B 0,C 180,E1 -571.453,E2 -571.453} C_VEL
LIN {X 0,Y 601.428,Z 166.381,A -85,B 0,C 180,E1 -574.117,E2 -574.117} C_VEL
LIN {X 0,Y 601.414,Z 166.383,A -85,B 0,C 180,E1 -576.581,E2 -576.581} C_VEL
LIN {X 0,Y 601.411,Z 166.385,A -85,B 0,C 180,E1 -579.532,E2 -579.532} C_VEL
LIN {X 0,Y 601.416,Z 166.383,A -85,B 0,C 180,E1 -581.765,E2 -581.765} C_VEL
LIN {X 0,Y 601.42,Z 166.383,A -85,B 0,C 180,E1 -584.534,E2 -584.534} C_VEL
LIN {X 0,Y 601.408,Z 166.388,A -85,B 0,C 180,E1 -587.408,E2 -587.408} C_VEL
LIN {X 0,Y 601.397,Z 166.39,A -85,B 0,C 180,E1 -590.003,E2 -590.003} C_VEL
LIN {X 0,Y 601.429,Z 166.385,A -85,B 0,C 180,E1 -592.617,E2 -592.617} C_VEL
LIN {X 0,Y 601.437,Z 166.384,A -85,B 0,C 180,E1 -595.069,E2 -595.069} C_VEL
LIN {X 0,Y 601.43,Z 166.383,A -85,B 0,C 180,E1 -597.484,E2 -597.484} C_VEL
LIN {X 0,Y 601.444,Z 166.38,A -85,B 0,C 180,E1 -599.847,E2 -599.847} C_VEL
LIN {X 0,Y 601.45,Z 166.382,A -85,B 0,C 180,E1 -602.889,E2 -602.889} C_VEL
LIN {X 0,Y 601.455,Z 166.378,A -85,B 0,C 180,E1 -605.859,E2 -605.859} C_VEL
LIN {X 0,Y 601.401,Z 166.385,A -85,B 0,C 180,E1 -608.76,E2 -608.76} C_VEL
LIN {X 0,Y 601.414,Z 166.386,A -85,B 0,C 180,E1 -611.608,E2 -611.608} C_VEL
LIN {X 0,Y 601.44,Z 166.38,A -85,B 0,C 180,E1 -613.713,E2 -613.713} C_VEL
LIN {X 0,Y 601.41,Z 166.384,A -85,B 0,C 180,E1 -616.484,E2 -616.484} C_VEL
LIN {X 0,Y 601.415,Z 166.386,A -85,B 0,C 180,E1 -619.224,E2 -619.224} C_VEL
LIN {X 0,Y 601.436,Z 166.385,A -85,B 0,C 180,E1 -621.939,E2 -621.939} C_VEL
LIN {X 0,Y 601.428,Z 166.384,A -85,B 0,C 180,E1 -624.636,E2 -624.636} C_VEL
LIN {X 0,Y 601.431,Z 166.382,A -85,B 0,C 180,E1 -627.321,E2 -627.321} C_VEL
LIN {X 0,Y 601.425,Z 166.382,A -85,B 0,C 180,E1 -630,E2 -630} C_VEL
LIN {X 0,Y 601.442,Z 166.38,A -85,B 0,C 180,E1 -632.679,E2 -632.679} C_VEL
LIN {X 0,Y 601.42,Z 166.382,A -85,B 0,C 180,E1 -635.364,E2 -635.364} C_VEL
LIN {X 0,Y 601.426,Z 166.382,A -85,B 0,C 180,E1 -638.061,E2 -638.061} C_VEL
LIN {X 0,Y 601.426,Z 166.385,A -85,B 0,C 180,E1 -641.018,E2 -641.018} C_VEL
LIN {X 0,Y 601.361,Z 166.393,A -85,B 0,C 180,E1 -643.517,E2 -643.517} C_VEL
LIN {X 0,Y 601.372,Z 171.226,A -85,B 0,C 180,E1 -646.289,E2 -646.289} C_VEL
LIN {X 0,Y 601.391,Z 175.776,A -85,B 0,C 180,E1 -648.815,E2 -648.815} C_VEL
LIN {X 0,Y 601.346,Z 180.16,A -85,B 0,C 180,E1 -651.241,E2 -651.241} C_VEL
LIN {X 0,Y 601.32,Z 184.232,A -85,B 0,C 180,E1 -653.414,E2 -653.414} C_VEL
LIN {X 0,Y 601.323,Z 188.871,A -85,B 0,C 180,E1 -655.852,E2 -655.852} C_VEL
LIN {X 0,Y 601.31,Z 194.514,A -85,B 0,C 180,E1 -658.769,E2 -658.769} C_VEL
LIN {X 0,Y 601.316,Z 199.754,A -85,B 0,C 180,E1 -661.44,E2 -661.44} C_VEL
LIN {X 0,Y 601.315,Z 205.082,A -85,B 0,C 180,E1 -664.126,E2 -664.126} C_VEL
LIN {X 0,Y 601.34,Z 209.884,A -85,B 0,C 180,E1 -666.442,E2 -666.442} C_VEL
LIN {X 0,Y 601.478,Z 219.879,A -85,B 0,C 180,E1 -666.734,E2 -666.734} C_VEL
LIN {X 0,Y 601.421,Z 229.019,A -85,B 0,C 180,E1 -667.105,E2 -667.105} C_VEL
LIN {X 0,Y 601.434,Z 238.815,A -85,B 0,C 180,E1 -667.63,E2 -667.63} C_VEL
LIN {X 0,Y 601.395,Z 247.773,A -85,B 0,C 180,E1 -668.27,E2 -668.27} C_VEL
LIN {X 0,Y 601.382,Z 255.339,A -85,B 0,C 180,E1 -668.95,E2 -668.95} C_VEL
LIN {X 0,Y 601.387,Z 262.387,A -85,B 0,C 180,E1 -669.738,E2 -669.738} C_VEL
LIN {X 0,Y 601.347,Z 268.178,A -85,B 0,C 180,E1 -670.567,E2 -670.567} C_VEL
LIN {X 0,Y 601.335,Z 271.91,A -85,B 0,C 180,E1 -671.233,E2 -671.233} C_VEL
LIN {X 0,Y 601.356,Z 275.904,A -85,B 0,C 180,E1 -672.176,E2 -672.176} C_VEL
LIN {X 0,Y 601.339,Z 277.597,A -85,B 0,C 180,E1 -672.677,E2 -672.677} C_VEL
LIN {X 0,Y 601.339,Z 279.717,A -85,B 0,C 180,E1 -673.594,E2 -673.594} C_VEL
LIN {X 0,Y 601.328,Z 280.784,A -85,B 0,C 180,E1 -674.527,E2 -674.527} C_VEL
LIN {X 0,Y 601.328,Z 280.825,A -85,B 0,C 180,E1 -675.474,E2 -675.474} C_VEL
LIN {X 0,Y 601.34,Z 279.802,A -85,B 0,C 180,E1 -676.436,E2 -676.436} C_VEL
LIN {X 0,Y 601.342,Z 277.588,A -85,B 0,C 180,E1 -677.417,E2 -677.417} C_VEL
LIN {X 0,Y 601.346,Z 273.911,A -85,B 0,C 180,E1 -678.415,E2 -678.415} C_VEL
LIN {X 0,Y 601.345,Z 268.681,A -85,B 0,C 180,E1 -679.435,E2 -679.435} C_VEL
LIN {X 0,Y 601.368,Z 263.099,A -85,B 0,C 180,E1 -680.263,E2 -680.263} C_VEL
LIN {X 0,Y 601.381,Z 256.232,A -85,B 0,C 180,E1 -681.051,E2 -681.051} C_VEL
LIN {X 0,Y 601.381,Z 248.854,A -85,B 0,C 180,E1 -681.73,E2 -681.73} C_VEL
LIN {X 0,Y 601.366,Z 240.258,A -85,B 0,C 180,E1 -682.366,E2 -682.366} C_VEL
LIN {X 0,Y 601.4,Z 229.858,A -85,B 0,C 180,E1 -682.948,E2 -682.948} C_VEL
LIN {X 0,Y 601.44,Z 221.013,A -85,B 0,C 180,E1 -683.317,E2 -683.317} C_VEL
LIN {X 0,Y 601.485,Z 211.971,A -85,B 0,C 180,E1 -683.593,E2 -683.593} C_VEL
LIN {X 0,Y 601.325,Z 209.697,A -85,B 0,C 180,E1 -683.658,E2 -683.658} C_VEL
LIN {X 0,Y 601.321,Z 204.851,A -85,B 0,C 180,E1 -686.08,E2 -686.08} C_VEL
LIN {X 0,Y 601.321,Z 199.929,A -85,B 0,C 180,E1 -688.561,E2 -688.561} C_VEL
LIN {X 0,Y 601.337,Z 194.418,A -85,B 0,C 180,E1 -691.369,E2 -691.369} C_VEL
LIN {X 0,Y 601.346,Z 189.046,A -85,B 0,C 180,E1 -694.146,E2 -694.146} C_VEL
LIN {X 0,Y 601.33,Z 184.399,A -85,B 0,C 180,E1 -696.587,E2 -696.587} C_VEL
LIN {X 0,Y 601.353,Z 179.035,A -85,B 0,C 180,E1 -699.476,E2 -699.476} C_VEL
LIN {X 0,Y 601.391,Z 173.938,A -85,B 0,C 180,E1 -702.312,E2 -702.312} C_VEL
LIN {X 0,Y 601.366,Z 168.967,A -85,B 0,C 180,E1 -705.102,E2 -705.102} C_VEL
LIN {X 0,Y 601.386,Z 166.464,A -85,B 0,C 180,E1 -706.484,E2 -706.484} C_VEL
LIN {X 0,Y 601.411,Z 166.385,A -85,B 0,C 180,E1 -709.224,E2 -709.224} C_VEL
LIN {X 0,Y 601.439,Z 166.382,A -85,B 0,C 180,E1 -711.94,E2 -711.94} C_VEL
LIN {X 0,Y 601.43,Z 166.384,A -85,B 0,C 180,E1 -714.637,E2 -714.637} C_VEL
LIN {X 0,Y 601.431,Z 166.382,A -85,B 0,C 180,E1 -717.322,E2 -717.322} C_VEL
LIN {X 0,Y 601.443,Z 166.382,A -85,B 0,C 180,E1 -720.001,E2 -720.001} C_VEL
LIN {X 0,Y 601.444,Z 166.382,A -85,B 0,C 180,E1 -722.68,E2 -722.68} C_VEL
LIN {X 0,Y 601.419,Z 166.383,A -85,B 0,C 180,E1 -725.365,E2 -725.365} C_VEL
LIN {X 0,Y 601.434,Z 166.383,A -85,B 0,C 180,E1 -728.061,E2 -728.061} C_VEL
LIN {X 0,Y 601.425,Z 166.383,A -85,B 0,C 180,E1 -731.012,E2 -731.012} C_VEL
LIN {X 0,Y 601.414,Z 166.384,A -85,B 0,C 180,E1 -733.516,E2 -733.516} C_VEL
LIN {X 0,Y 601.44,Z 166.384,A -85,B 0,C 180,E1 -736.287,E2 -736.287} C_VEL
LIN {X 0,Y 601.418,Z 166.383,A -85,B 0,C 180,E1 -739.099,E2 -739.099} C_VEL
LIN {X 0,Y 601.406,Z 166.385,A -85,B 0,C 180,E1 -741.24,E2 -741.24} C_VEL
LIN {X 0,Y 601.463,Z 166.38,A -85,B 0,C 180,E1 -744.14,E2 -744.14} C_VEL
LIN {X 0,Y 601.44,Z 166.381,A -85,B 0,C 180,E1 -747.112,E2 -747.112} C_VEL
LIN {X 0,Y 601.425,Z 166.383,A -85,B 0,C 180,E1 -749.393,E2 -749.393} C_VEL
LIN {X 0,Y 601.412,Z 166.384,A -85,B 0,C 180,E1 -751.727,E2 -751.727} C_VEL
LIN {X 0,Y 601.432,Z 166.382,A -85,B 0,C 180,E1 -754.118,E2 -754.118} C_VEL
LIN {X 0,Y 601.439,Z 166.381,A -85,B 0,C 180,E1 -757.382,E2 -757.382} C_VEL
LIN {X 0,Y 601.403,Z 166.386,A -85,B 0,C 180,E1 -759.996,E2 -759.996} C_VEL
LIN {X 0,Y 601.41,Z 166.388,A -85,B 0,C 180,E1 -762.671,E2 -762.671} C_VEL
LIN {X 0,Y 601.428,Z 166.382,A -85,B 0,C 180,E1 -765.482,E2 -765.482} C_VEL
LIN {X 0,Y 601.423,Z 166.386,A -85,B 0,C 180,E1 -768.407,E2 -768.407} C_VEL
LIN {X 0,Y 601.438,Z 166.382,A -85,B 0,C 180,E1 -771.529,E2 -771.529} C_VEL
LIN {X 0,Y 601.391,Z 166.389,A -85,B 0,C 180,E1 -774.246,E2 -774.246} C_VEL
LIN {X 0,Y 601.429,Z 166.384,A -85,B 0,C 180,E1 -776.687,E2 -776.687} C_VEL
LIN {X 0,Y 601.453,Z 166.452,A -85,B 0,C 180,E1 -779.167,E2 -779.167} C_VEL
LIN {X 0,Y 601.506,Z 174.128,A -85,B 0,C 180,E1 -781.377,E2 -781.377} C_VEL
LIN {X 0,Y 601.466,Z 184.306,A -85,B 0,C 180,E1 -784.122,E2 -784.122} C_VEL
LIN {X 0,Y 601.42,Z 194.955,A -85,B 0,C 180,E1 -786.954,E2 -786.954} C_VEL
LIN {X 0,Y 601.414,Z 204.635,A -85,B 0,C 180,E1 -789.478,E2 -789.478} C_VEL
LIN {X 0,Y 601.425,Z 215.697,A -85,B 0,C 180,E1 -792.313,E2 -792.313} C_VEL
LIN {X 0,Y 601.366,Z 226.759,A -85,B 0,C 180,E1 -795.102,E2 -795.102} C_VEL
LIN {X 0,Y 601.365,Z 237.821,A -85,B 0,C 180,E1 -797.857,E2 -797.857} C_VEL
LIN {X 0,Y 601.367,Z 249.097,A -85,B 0,C 180,E1 -800.594,E2 -800.594} C_VEL
LIN {X 0,Y 601.514,Z 259.738,A -85,B 0,C 180,E1 -800.84,E2 -800.84} C_VEL
LIN {X 0,Y 601.447,Z 271.538,A -85,B 0,C 180,E1 -801.263,E2 -801.263} C_VEL
LIN {X 0,Y 601.423,Z 280.237,A -85,B 0,C 180,E1 -801.685,E2 -801.685} C_VEL
LIN {X 0,Y 601.428,Z 288.545,A -85,B 0,C 180,E1 -802.193,E2 -802.193} C_VEL
LIN {X 0,Y 601.414,Z 296.403,A -85,B 0,C 180,E1 -802.783,E2 -802.783} C_VEL
LIN {X 0,Y 601.412,Z 303.599,A -85,B 0,C 180,E1 -803.443,E2 -803.443} C_VEL
LIN {X 0,Y 601.391,Z 311.192,A -85,B 0,C 180,E1 -804.299,E2 -804.299} C_VEL
LIN {X 0,Y 601.38,Z 317.028,A -85,B 0,C 180,E1 -805.14,E2 -805.14} C_VEL
LIN {X 0,Y 601.345,Z 321.631,A -85,B 0,C 180,E1 -805.979,E2 -805.979} C_VEL
LIN {X 0,Y 601.343,Z 324.622,A -85,B 0,C 180,E1 -806.65,E2 -806.65} C_VEL
LIN {X 0,Y 601.326,Z 326.932,A -85,B 0,C 180,E1 -807.321,E2 -807.321} C_VEL
LIN {X 0,Y 601.343,Z 328.679,A -85,B 0,C 180,E1 -807.991,E2 -807.991} C_VEL
LIN {X 0,Y 601.345,Z 329.935,A -85,B 0,C 180,E1 -808.661,E2 -808.661} C_VEL
LIN {X 0,Y 601.335,Z 330.713,A -85,B 0,C 180,E1 -809.33,E2 -809.33} C_VEL
LIN {X 0,Y 601.332,Z 331,A -85,B 0,C 180,E1 -810,E2 -810} C_VEL
LIN {X 0,Y 601.335,Z 330.713,A -85,B 0,C 180,E1 -810.67,E2 -810.67} C_VEL
LIN {X 0,Y 601.345,Z 329.934,A -85,B 0,C 180,E1 -811.339,E2 -811.339} C_VEL
LIN {X 0,Y 601.343,Z 328.678,A -85,B 0,C 180,E1 -812.009,E2 -812.009} C_VEL
LIN {X 0,Y 601.342,Z 325.786,A -85,B 0,C 180,E1 -813.015,E2 -813.015} C_VEL
LIN {X 0,Y 601.364,Z 323.146,A -85,B 0,C 180,E1 -813.685,E2 -813.685} C_VEL
LIN {X 0,Y 601.341,Z 317.984,A -85,B 0,C 180,E1 -814.693,E2 -814.693} C_VEL
LIN {X 0,Y 601.383,Z 312.429,A -85,B 0,C 180,E1 -815.533,E2 -815.533} C_VEL
LIN {X 0,Y 601.393,Z 305.154,A -85,B 0,C 180,E1 -816.403,E2 -816.403} C_VEL
LIN {X 0,Y 601.417,Z 297.414,A -85,B 0,C 180,E1 -817.132,E2 -817.132} C_VEL
LIN {X 0,Y 601.436,Z 289.76,A -85,B 0,C 180,E1 -817.723,E2 -817.723} C_VEL
LIN {X 0,Y 601.433,Z 281.72,A -85,B 0,C 180,E1 -818.23,E2 -818.23} C_VEL
LIN {X 0,Y 601.457,Z 273.389,A -85,B 0,C 180,E1 -818.653,E2 -818.653} C_VEL
LIN {X 0,Y 601.469,Z 264.885,A -85,B 0,C 180,E1 -818.991,E2 -818.991} C_VEL
LIN {X 0,Y 601.483,Z 254.748,A -85,B 0,C 180,E1 -819.288,E2 -819.288} C_VEL
LIN {X 0,Y 601.342,Z 248.882,A -85,B 0,C 180,E1 -819.417,E2 -819.417} C_VEL
LIN {X 0,Y 601.365,Z 237.82,A -85,B 0,C 180,E1 -822.144,E2 -822.144} C_VEL
LIN {X 0,Y 601.366,Z 226.758,A -85,B 0,C 180,E1 -824.899,E2 -824.899} C_VEL
LIN {X 0,Y 601.425,Z 215.696,A -85,B 0,C 180,E1 -827.688,E2 -827.688} C_VEL
LIN {X 0,Y 601.414,Z 204.634,A -85,B 0,C 180,E1 -830.523,E2 -830.523} C_VEL
LIN {X 0,Y 601.466,Z 193.572,A -85,B 0,C 180,E1 -833.409,E2 -833.409} C_VEL
LIN {X 0,Y 601.464,Z 184.296,A -85,B 0,C 180,E1 -835.877,E2 -835.877} C_VEL
LIN {X 0,Y 601.519,Z 174.224,A -85,B 0,C 180,E1 -838.623,E2 -838.623} C_VEL
LIN {X 0,Y 601.449,Z 166.451,A -85,B 0,C 180,E1 -840.819,E2 -840.819} C_VEL
LIN {X 0,Y 601.418,Z 166.383,A -85,B 0,C 180,E1 -843.314,E2 -843.314} C_VEL
LIN {X 0,Y 601.397,Z 166.386,A -85,B 0,C 180,E1 -846.26,E2 -846.26} C_VEL
LIN {X 0,Y 601.436,Z 166.38,A -85,B 0,C 180,E1 -848.471,E2 -848.471} C_VEL
LIN {X 0,Y 601.422,Z 166.385,A -85,B 0,C 180,E1 -851.593,E2 -851.593} C_VEL
LIN {X 0,Y 601.429,Z 166.382,A -85,B 0,C 180,E1 -854.535,E2 -854.535} C_VEL
LIN {X 0,Y 601.387,Z 166.386,A -85,B 0,C 180,E1 -857.327,E2 -857.327} C_VEL
LIN {X 0,Y 601.401,Z 166.385,A -85,B 0,C 180,E1 -860.004,E2 -860.004} C_VEL
LIN {X 0,Y 601.441,Z 166.38,A -85,B 0,C 180,E1 -862.618,E2 -862.618} C_VEL
LIN {X 0,Y 601.429,Z 166.384,A -85,B 0,C 180,E1 -865.881,E2 -865.881} C_VEL
LIN {X 0,Y 601.42,Z 166.384,A -85,B 0,C 180,E1 -868.546,E2 -868.546} C_VEL
LIN {X 0,Y 601.414,Z 166.383,A -85,B 0,C 180,E1 -871.372,E2 -871.372} C_VEL
LIN {X 0,Y 601.42,Z 166.382,A -85,B 0,C 180,E1 -874.132,E2 -874.132} C_VEL
LIN {X 0,Y 601.402,Z 166.385,A -85,B 0,C 180,E1 -876.589,E2 -876.589} C_VEL
LIN {X 0,Y 601.424,Z 166.383,A -85,B 0,C 180,E1 -879.478,E2 -879.478} C_VEL
LIN {X 0,Y 601.393,Z 166.39,A -85,B 0,C 180,E1 -882.311,E2 -882.311} C_VEL
LIN {X 0,Y 601.42,Z 166.383,A -85,B 0,C 180,E1 -884.408,E2 -884.408} C_VEL
LIN {X 0,Y 601.417,Z 166.384,A -85,B 0,C 180,E1 -887.171,E2 -887.171} C_VEL
LIN {X 0,Y 601.429,Z 166.385,A -85,B 0,C 180,E1 -889.904,E2 -889.904} C_VEL
LIN {X 0,Y 601.412,Z 166.387,A -85,B 0,C 180,E1 -892.614,E2 -892.614} C_VEL
LIN {X 0,Y 601.427,Z 166.383,A -85,B 0,C 180,E1 -895.308,E2 -895.308} C_VEL
LIN {X 0,Y 601.41,Z 166.384,A -85,B 0,C 180,E1 -897.99,E2 -897.99} C_VEL
LIN {X 0,Y 601.437,Z 166.381,A -85,B 0,C 180,E1 -900.669,E2 -900.669} C_VEL
LIN {X 0,Y 601.433,Z 166.381,A -85,B 0,C 180,E1 -903.349,E2 -903.349} C_VEL
LIN {X 0,Y 601.398,Z 166.385,A -85,B 0,C 180,E1 -906.037,E2 -906.037} C_VEL
LIN {X 0,Y 601.438,Z 166.382,A -85,B 0,C 180,E1 -908.06,E2 -908.06} C_VEL
LIN {X 0,Y 601.43,Z 166.381,A -85,B 0,C 180,E1 -911.013,E2 -911.013} C_VEL
LIN {X 0,Y 601.402,Z 166.385,A -85,B 0,C 180,E1 -912.372,E2 -912.372} C_VEL
LIN {X 0,Y 600.736,Z 166.472,A -85,B 0,C 180,E1 -912.932,E2 -912.932} C_VEL
LIN {X 0,Y 597.892,Z 166.823,A -85,B 0,C 180,E1 -913.84,E2 -913.84} C_VEL
LIN {X 0,Y 595.486,Z 167.123,A -85,B 0,C 180,E1 -914.57,E2 -914.57} C_VEL
LIN {X 0,Y 594.448,Z 167.252,A -85,B 0,C 180,E1 -915.134,E2 -915.134} C_VEL
LIN {X 0,Y 594.36,Z 167.261,A -85,B 0,C 180,E1 -915.324,E2 -915.324} C_VEL
LIN {X 0,Y 594.352,Z 167.265,A -85,B 0,C 180,E1 -917.904,E2 -917.904} C_VEL
LIN {X 0,Y 594.406,Z 167.259,A -85,B 0,C 180,E1 -920.775,E2 -920.775} C_VEL
LIN {X 0,Y 594.37,Z 167.261,A -85,B 0,C 180,E1 -923.704,E2 -923.704} C_VEL
LIN {X 0,Y 594.391,Z 167.259,A -85,B 0,C 180,E1 -926.023,E2 -926.023} C_VEL
LIN {X 0,Y 594.384,Z 167.259,A -85,B 0,C 180,E1 -928.997,E2 -928.997} C_VEL
LIN {X 0,Y 594.375,Z 167.26,A -85,B 0,C 180,E1 -931.642,E2 -931.642} C_VEL
LIN {X 0,Y 594.38,Z 167.263,A -85,B 0,C 180,E1 -934.579,E2 -934.579} C_VEL
LIN {X 0,Y 594.385,Z 167.261,A -85,B 0,C 180,E1 -937.086,E2 -937.086} C_VEL
LIN {X 0,Y 594.357,Z 167.266,A -85,B 0,C 180,E1 -939.772,E2 -939.772} C_VEL
LIN {X 0,Y 594.366,Z 167.265,A -85,B 0,C 180,E1 -942.374,E2 -942.374} C_VEL
LIN {X 0,Y 594.359,Z 167.263,A -85,B 0,C 180,E1 -945.19,E2 -945.19} C_VEL
LIN {X 0,Y 594.382,Z 167.259,A -85,B 0,C 180,E1 -948.15,E2 -948.15} C_VEL
LIN {X 0,Y 594.379,Z 167.264,A -85,B 0,C 180,E1 -951.295,E2 -951.295} C_VEL
LIN {X 0,Y 594.387,Z 167.262,A -85,B 0,C 180,E1 -953.758,E2 -953.758} C_VEL
LIN {X 0,Y 594.38,Z 167.262,A -85,B 0,C 180,E1 -956.239,E2 -956.239} C_VEL
LIN {X 0,Y 594.386,Z 167.26,A -85,B 0,C 180,E1 -958.65,E2 -958.65} C_VEL
LIN {X 0,Y 594.378,Z 167.26,A -85,B 0,C 180,E1 -961.041,E2 -961.041} C_VEL
LIN {X 0,Y 594.379,Z 167.263,A -85,B 0,C 180,E1 -963.976,E2 -963.976} C_VEL
LIN {X 0,Y 594.387,Z 167.26,A -85,B 0,C 180,E1 -966.296,E2 -966.296} C_VEL
LIN {X 0,Y 594.406,Z 167.26,A -85,B 0,C 180,E1 -969.224,E2 -969.224} C_VEL
LIN {X 0,Y 594.344,Z 167.264,A -85,B 0,C 180,E1 -972.094,E2 -972.094} C_VEL
LIN {X 0,Y 594.363,Z 167.265,A -85,B 0,C 180,E1 -974.219,E2 -974.219} C_VEL
LIN {X 0,Y 594.37,Z 167.263,A -85,B 0,C 180,E1 -977.017,E2 -977.017} C_VEL
LIN {X 0,Y 594.381,Z 167.259,A -85,B 0,C 180,E1 -979.784,E2 -979.784} C_VEL
LIN {X 0,Y 594.363,Z 167.261,A -85,B 0,C 180,E1 -982.526,E2 -982.526} C_VEL
LIN {X 0,Y 594.395,Z 167.258,A -85,B 0,C 180,E1 -985.252,E2 -985.252} C_VEL
LIN {X 0,Y 594.382,Z 167.26,A -85,B 0,C 180,E1 -987.967,E2 -987.967} C_VEL
LIN {X 0,Y 594.415,Z 167.257,A -85,B 0,C 180,E1 -990.677,E2 -990.677} C_VEL
LIN {X 0,Y 594.382,Z 167.263,A -85,B 0,C 180,E1 -993.389,E2 -993.389} C_VEL
LIN {X 0,Y 594.371,Z 167.263,A -85,B 0,C 180,E1 -996.109,E2 -996.109} C_VEL
LIN {X 0,Y 594.396,Z 167.258,A -85,B 0,C 180,E1 -998.842,E2 -998.842} C_VEL
LIN {X 0,Y 594.385,Z 167.259,A -85,B 0,C 180,E1 -1001.596,E2 -1001.596} C_VEL
LIN {X 0,Y 594.296,Z 167.332,A -85,B 0,C 180,E1 -1003.681,E2 -1003.681} C_VEL
LIN {X 0,Y 594.314,Z 172.28,A -85,B 0,C 180,E1 -1006.488,E2 -1006.488} C_VEL
LIN {X 0,Y 594.307,Z 177.383,A -85,B 0,C 180,E1 -1009.336,E2 -1009.336} C_VEL
LIN {X 0,Y 594.269,Z 181.284,A -85,B 0,C 180,E1 -1011.507,E2 -1011.507} C_VEL
LIN {X 0,Y 594.243,Z 185.289,A -85,B 0,C 180,E1 -1013.71,E2 -1013.71} C_VEL
LIN {X 0,Y 594.223,Z 190.948,A -85,B 0,C 180,E1 -1016.707,E2 -1016.707} C_VEL
LIN {X 0,Y 594.234,Z 195.354,A -85,B 0,C 180,E1 -1019.006,E2 -1019.006} C_VEL
LIN {X 0,Y 594.222,Z 200.428,A -85,B 0,C 180,E1 -1021.62,E2 -1021.62} C_VEL
LIN {X 0,Y 594.24,Z 205.331,A -85,B 0,C 180,E1 -1024.12,E2 -1024.12} C_VEL
LIN {X 0,Y 594.258,Z 209.73,A -85,B 0,C 180,E1 -1026.335,E2 -1026.335} C_VEL
LIN {X 0,Y 594.447,Z 218.915,A -85,B 0,C 180,E1 -1026.601,E2 -1026.601} C_VEL
LIN {X 0,Y 594.391,Z 227.639,A -85,B 0,C 180,E1 -1026.946,E2 -1026.946} C_VEL
LIN {X 0,Y 594.393,Z 235.84,A -85,B 0,C 180,E1 -1027.369,E2 -1027.369} C_VEL
LIN {X 0,Y 594.371,Z 244.612,A -85,B 0,C 180,E1 -1027.942,E2 -1027.942} C_VEL
LIN {X 0,Y 594.327,Z 253.559,A -85,B 0,C 180,E1 -1028.699,E2 -1028.699} C_VEL
LIN {X 0,Y 594.316,Z 260.645,A -85,B 0,C 180,E1 -1029.465,E2 -1029.465} C_VEL
LIN {X 0,Y 594.288,Z 265.753,A -85,B 0,C 180,E1 -1030.146,E2 -1030.146} C_VEL
LIN {X 0,Y 594.263,Z 271.559,A -85,B 0,C 180,E1 -1031.117,E2 -1031.117} C_VEL
LIN {X 0,Y 594.268,Z 274.811,A -85,B 0,C 180,E1 -1031.837,E2 -1031.837} C_VEL
LIN {X 0,Y 594.248,Z 278.092,A -85,B 0,C 180,E1 -1032.842,E2 -1032.842} C_VEL
LIN {X 0,Y 594.231,Z 280.067,A -85,B 0,C 180,E1 -1033.827,E2 -1033.827} C_VEL
LIN {X 0,Y 594.214,Z 280.91,A -85,B 0,C 180,E1 -1034.796,E2 -1034.796} C_VEL
LIN {X 0,Y 594.225,Z 280.698,A -85,B 0,C 180,E1 -1035.75,E2 -1035.75} C_VEL
LIN {X 0,Y 594.241,Z 279.406,A -85,B 0,C 180,E1 -1036.69,E2 -1036.69} C_VEL
LIN {X 0,Y 594.268,Z 277.023,A -85,B 0,C 180,E1 -1037.617,E2 -1037.617} C_VEL
LIN {X 0,Y 594.242,Z 273.599,A -85,B 0,C 180,E1 -1038.526,E2 -1038.526} C_VEL
LIN {X 0,Y 594.264,Z 269.027,A -85,B 0,C 180,E1 -1039.426,E2 -1039.426} C_VEL
LIN {X 0,Y 594.306,Z 263.172,A -85,B 0,C 180,E1 -1040.315,E2 -1040.315} C_VEL
LIN {X 0,Y 594.328,Z 255.544,A -85,B 0,C 180,E1 -1041.192,E2 -1041.192} C_VEL
LIN {X 0,Y 594.324,Z 247.206,A -85,B 0,C 180,E1 -1041.948,E2 -1041.948} C_VEL
LIN {X 0,Y 594.351,Z 237.409,A -85,B 0,C 180,E1 -1042.631,E2 -1042.631} C_VEL
LIN {X 0,Y 594.378,Z 228.651,A -85,B 0,C 180,E1 -1043.097,E2 -1043.097} C_VEL
LIN {X 0,Y 594.44,Z 220.053,A -85,B 0,C 180,E1 -1043.449,E2 -1043.449} C_VEL
LIN {X 0,Y 594.39,Z 211.234,A -85,B 0,C 180,E1 -1043.714,E2 -1043.714} C_VEL
LIN {X 0,Y 594.235,Z 209.671,A -85,B 0,C 180,E1 -1043.775,E2 -1043.775} C_VEL
LIN {X 0,Y 594.234,Z 204.818,A -85,B 0,C 180,E1 -1046.231,E2 -1046.231} C_VEL
LIN {X 0,Y 594.243,Z 200.088,A -85,B 0,C 180,E1 -1048.643,E2 -1048.643} C_VEL
LIN {X 0,Y 594.251,Z 195.389,A -85,B 0,C 180,E1 -1051.065,E2 -1051.065} C_VEL
LIN {X 0,Y 594.25,Z 191.113,A -85,B 0,C 180,E1 -1053.295,E2 -1053.295} C_VEL
LIN {X 0,Y 594.25,Z 185.455,A -85,B 0,C 180,E1 -1056.291,E2 -1056.291} C_VEL
LIN {X 0,Y 594.255,Z 181.469,A -85,B 0,C 180,E1 -1058.493,E2 -1058.493} C_VEL
LIN {X 0,Y 594.311,Z 176.324,A -85,B 0,C 180,E1 -1061.381,E2 -1061.381} C_VEL
LIN {X 0,Y 594.305,Z 171.285,A -85,B 0,C 180,E1 -1064.218,E2 -1064.218} C_VEL
LIN {X 0,Y 594.327,Z 167.509,A -85,B 0,C 180,E1 -1066.321,E2 -1066.321} C_VEL
LIN {X 0,Y 594.394,Z 167.259,A -85,B 0,C 180,E1 -1068.405,E2 -1068.405} C_VEL
LIN {X 0,Y 594.38,Z 167.263,A -85,B 0,C 180,E1 -1071.159,E2 -1071.159} C_VEL
LIN {X 0,Y 594.361,Z 167.263,A -85,B 0,C 180,E1 -1073.892,E2 -1073.892} C_VEL
LIN {X 0,Y 594.385,Z 167.262,A -85,B 0,C 180,E1 -1076.611,E2 -1076.611} C_VEL
LIN {X 0,Y 594.417,Z 167.257,A -85,B 0,C 180,E1 -1079.323,E2 -1079.323} C_VEL
LIN {X 0,Y 594.387,Z 167.259,A -85,B 0,C 180,E1 -1082.033,E2 -1082.033} C_VEL
LIN {X 0,Y 594.397,Z 167.261,A -85,B 0,C 180,E1 -1084.748,E2 -1084.748} C_VEL
LIN {X 0,Y 594.395,Z 167.259,A -85,B 0,C 180,E1 -1087.474,E2 -1087.474} C_VEL
LIN {X 0,Y 594.393,Z 167.259,A -85,B 0,C 180,E1 -1090.216,E2 -1090.216} C_VEL
LIN {X 0,Y 594.366,Z 167.264,A -85,B 0,C 180,E1 -1092.984,E2 -1092.984} C_VEL
LIN {X 0,Y 594.374,Z 167.264,A -85,B 0,C 180,E1 -1095.078,E2 -1095.078} C_VEL
LIN {X 0,Y 594.383,Z 167.261,A -85,B 0,C 180,E1 -1097.194,E2 -1097.194} C_VEL
LIN {X 0,Y 594.375,Z 167.261,A -85,B 0,C 180,E1 -1100.054,E2 -1100.054} C_VEL
LIN {X 0,Y 594.36,Z 167.264,A -85,B 0,C 180,E1 -1102.968,E2 -1102.968} C_VEL
LIN {X 0,Y 594.378,Z 167.262,A -85,B 0,C 180,E1 -1105.193,E2 -1105.193} C_VEL
LIN {X 0,Y 594.37,Z 167.263,A -85,B 0,C 180,E1 -1107.524,E2 -1107.524} C_VEL
LIN {X 0,Y 594.388,Z 167.26,A -85,B 0,C 180,E1 -1110.328,E2 -1110.328} C_VEL
LIN {X 0,Y 594.38,Z 167.26,A -85,B 0,C 180,E1 -1112.95,E2 -1112.95} C_VEL
LIN {X 0,Y 594.355,Z 167.264,A -85,B 0,C 180,E1 -1115.409,E2 -1115.409} C_VEL
LIN {X 0,Y 594.387,Z 167.262,A -85,B 0,C 180,E1 -1117.941,E2 -1117.941} C_VEL
LIN {X 0,Y 594.377,Z 167.261,A -85,B 0,C 180,E1 -1120.822,E2 -1120.822} C_VEL
LIN {X 0,Y 594.37,Z 167.264,A -85,B 0,C 180,E1 -1123.84,E2 -1123.84} C_VEL
LIN {X 0,Y 594.366,Z 167.262,A -85,B 0,C 180,E1 -1126.7,E2 -1126.7} C_VEL
LIN {X 0,Y 594.369,Z 167.265,A -85,B 0,C 180,E1 -1129.433,E2 -1129.433} C_VEL
LIN {X 0,Y 594.391,Z 167.259,A -85,B 0,C 180,E1 -1132.392,E2 -1132.392} C_VEL
LIN {X 0,Y 594.399,Z 167.261,A -85,B 0,C 180,E1 -1135.421,E2 -1135.421} C_VEL
LIN {X 0,Y 594.378,Z 167.262,A -85,B 0,C 180,E1 -1138.358,E2 -1138.358} C_VEL
LIN {X 0,Y 594.428,Z 167.468,A -85,B 0,C 180,E1 -1139.049,E2 -1139.049} C_VEL
LIN {X 0,Y 594.562,Z 174.162,A -85,B 0,C 180,E1 -1141.011,E2 -1141.011} C_VEL
LIN {X 0,Y 594.451,Z 182.44,A -85,B 0,C 180,E1 -1143.304,E2 -1143.304} C_VEL
LIN {X 0,Y 594.454,Z 192.19,A -85,B 0,C 180,E1 -1145.928,E2 -1145.928} C_VEL
LIN {X 0,Y 594.396,Z 203.144,A -85,B 0,C 180,E1 -1148.833,E2 -1148.833} C_VEL
LIN {X 0,Y 594.369,Z 212.931,A -85,B 0,C 180,E1 -1151.382,E2 -1151.382} C_VEL
LIN {X 0,Y 594.329,Z 223.993,A -85,B 0,C 180,E1 -1154.218,E2 -1154.218} C_VEL
LIN {X 0,Y 594.3,Z 235.056,A -85,B 0,C 180,E1 -1157.016,E2 -1157.016} C_VEL
LIN {X 0,Y 594.275,Z 246.118,A -85,B 0,C 180,E1 -1159.782,E2 -1159.782} C_VEL
LIN {X 0,Y 594.3,Z 249.095,A -85,B 0,C 180,E1 -1160.481,E2 -1160.481} C_VEL
LIN {X 0,Y 594.505,Z 256.417,A -85,B 0,C 180,E1 -1160.645,E2 -1160.645} C_VEL
LIN {X 0,Y 594.458,Z 264.893,A -85,B 0,C 180,E1 -1160.902,E2 -1160.902} C_VEL
LIN {X 0,Y 594.423,Z 273.398,A -85,B 0,C 180,E1 -1161.244,E2 -1161.244} C_VEL
LIN {X 0,Y 594.411,Z 281.727,A -85,B 0,C 180,E1 -1161.672,E2 -1161.672} C_VEL
LIN {X 0,Y 594.371,Z 289.765,A -85,B 0,C 180,E1 -1162.185,E2 -1162.185} C_VEL
LIN {X 0,Y 594.358,Z 297.417,A -85,B 0,C 180,E1 -1162.783,E2 -1162.783} C_VEL
LIN {X 0,Y 594.33,Z 305.812,A -85,B 0,C 180,E1 -1163.59,E2 -1163.59} C_VEL
LIN {X 0,Y 594.309,Z 312.432,A -85,B 0,C 180,E1 -1164.401,E2 -1164.401} C_VEL
LIN {X 0,Y 594.256,Z 317.987,A -85,B 0,C 180,E1 -1165.251,E2 -1165.251} C_VEL
LIN {X 0,Y 594.286,Z 323.147,A -85,B 0,C 180,E1 -1166.271,E2 -1166.271} C_VEL
LIN {X 0,Y 594.245,Z 325.788,A -85,B 0,C 180,E1 -1166.949,E2 -1166.949} C_VEL
LIN {X 0,Y 594.242,Z 328.68,A -85,B 0,C 180,E1 -1167.967,E2 -1167.967} C_VEL
LIN {X 0,Y 594.245,Z 329.935,A -85,B 0,C 180,E1 -1168.645,E2 -1168.645} C_VEL
LIN {X 0,Y 594.235,Z 330.713,A -85,B 0,C 180,E1 -1169.322,E2 -1169.322} C_VEL
LIN {X 0,Y 594.233,Z 331,A -85,B 0,C 180,E1 -1170,E2 -1170} C_VEL
LIN {X 0,Y 594.235,Z 330.712,A -85,B 0,C 180,E1 -1170.678,E2 -1170.678} C_VEL
LIN {X 0,Y 594.245,Z 329.935,A -85,B 0,C 180,E1 -1171.356,E2 -1171.356} C_VEL
LIN {X 0,Y 594.242,Z 328.679,A -85,B 0,C 180,E1 -1172.033,E2 -1172.033} C_VEL
LIN {X 0,Y 594.245,Z 325.787,A -85,B 0,C 180,E1 -1173.051,E2 -1173.051} C_VEL
LIN {X 0,Y 594.286,Z 323.146,A -85,B 0,C 180,E1 -1173.729,E2 -1173.729} C_VEL
LIN {X 0,Y 594.256,Z 317.984,A -85,B 0,C 180,E1 -1174.749,E2 -1174.749} C_VEL
LIN {X 0,Y 594.319,Z 311.188,A -85,B 0,C 180,E1 -1175.769,E2 -1175.769} C_VEL
LIN {X 0,Y 594.343,Z 303.514,A -85,B 0,C 180,E1 -1176.644,E2 -1176.644} C_VEL
LIN {X 0,Y 594.355,Z 296.402,A -85,B 0,C 180,E1 -1177.303,E2 -1177.303} C_VEL
LIN {X 0,Y 594.393,Z 288.545,A -85,B 0,C 180,E1 -1177.901,E2 -1177.901} C_VEL
LIN {X 0,Y 594.419,Z 278.734,A -85,B 0,C 180,E1 -1178.499,E2 -1178.499} C_VEL
LIN {X 0,Y 594.465,Z 267.293,A -85,B 0,C 180,E1 -1179.012,E2 -1179.012} C_VEL
LIN {X 0,Y 594.494,Z 257.239,A -85,B 0,C 180,E1 -1179.334,E2 -1179.334} C_VEL
LIN {X 0,Y 594.27,Z 248.882,A -85,B 0,C 180,E1 -1179.53,E2 -1179.53} C_VEL
LIN {X 0,Y 594.318,Z 237.82,A -85,B 0,C 180,E1 -1182.29,E2 -1182.29} C_VEL
LIN {X 0,Y 594.317,Z 226.758,A -85,B 0,C 180,E1 -1185.08,E2 -1185.08} C_VEL
LIN {X 0,Y 594.376,Z 215.696,A -85,B 0,C 180,E1 -1187.905,E2 -1187.905} C_VEL
LIN {X 0,Y 594.387,Z 204.634,A -85,B 0,C 180,E1 -1190.776,E2 -1190.776} C_VEL
LIN {X 0,Y 594.448,Z 193.572,A -85,B 0,C 180,E1 -1193.702,E2 -1193.702} C_VEL
LIN {X 0,Y 594.441,Z 183.689,A -85,B 0,C 180,E1 -1196.326,E2 -1196.326} C_VEL
LIN {X 0,Y 594.564,Z 174.231,A -85,B 0,C 180,E1 -1198.989,E2 -1198.989} C_VEL
LIN {X 0,Y 594.594,Z 168.787,A -85,B 0,C 180,E1 -1200.548,E2 -1200.548} C_VEL
LIN {X 0,Y 594.387,Z 167.262,A -85,B 0,C 180,E1 -1201.053,E2 -1201.053} C_VEL
LIN {X 0,Y 594.378,Z 167.262,A -85,B 0,C 180,E1 -1203.762,E2 -1203.762} C_VEL
LIN {X 0,Y 594.372,Z 167.264,A -85,B 0,C 180,E1 -1206.481,E2 -1206.481} C_VEL
LIN {X 0,Y 594.382,Z 167.26,A -85,B 0,C 180,E1 -1208.805,E2 -1208.805} C_VEL
LIN {X 0,Y 594.379,Z 167.262,A -85,B 0,C 180,E1 -1211.848,E2 -1211.848} C_VEL
LIN {X 0,Y 594.359,Z 167.262,A -85,B 0,C 180,E1 -1214.808,E2 -1214.808} C_VEL
LIN {X 0,Y 594.351,Z 167.263,A -85,B 0,C 180,E1 -1217.623,E2 -1217.623} C_VEL
LIN {X 0,Y 594.368,Z 167.262,A -85,B 0,C 180,E1 -1220.319,E2 -1220.319} C_VEL
LIN {X 0,Y 594.386,Z 167.26,A -85,B 0,C 180,E1 -1222.913,E2 -1222.913} C_VEL
LIN {X 0,Y 594.382,Z 167.262,A -85,B 0,C 180,E1 -1225.862,E2 -1225.862} C_VEL
LIN {X 0,Y 594.37,Z 167.261,A -85,B 0,C 180,E1 -1228.649,E2 -1228.649} C_VEL
LIN {X 0,Y 594.38,Z 167.261,A -85,B 0,C 180,E1 -1231.043,E2 -1231.043} C_VEL
LIN {X 0,Y 594.393,Z 167.258,A -85,B 0,C 180,E1 -1233.977,E2 -1233.977} C_VEL
LIN {X 0,Y 594.374,Z 167.261,A -85,B 0,C 180,E1 -1236.295,E2 -1236.295} C_VEL
LIN {X 0,Y 594.397,Z 167.257,A -85,B 0,C 180,E1 -1239.224,E2 -1239.224} C_VEL
LIN {X 0,Y 594.353,Z 167.265,A -85,B 0,C 180,E1 -1242.095,E2 -1242.095} C_VEL
LIN {X 0,Y 594.373,Z 167.26,A -85,B 0,C 180,E1 -1244.219,E2 -1244.219} C_VEL
LIN {X 0,Y 594.379,Z 167.262,A -85,B 0,C 180,E1 -1246.321,E2 -1246.321} C_VEL
LIN {X 0,Y 594.372,Z 167.261,A -85,B 0,C 180,E1 -1249.094,E2 -1249.094} C_VEL
LIN {X 0,Y 594.387,Z 167.258,A -85,B 0,C 180,E1 -1251.842,E2 -1251.842} C_VEL
LIN {X 0,Y 594.381,Z 167.259,A -85,B 0,C 180,E1 -1254.572,E2 -1254.572} C_VEL
LIN {X 0,Y 594.406,Z 167.257,A -85,B 0,C 180,E1 -1257.289,E2 -1257.289} C_VEL
LIN {X 0,Y 594.419,Z 167.257,A -85,B 0,C 180,E1 -1259.999,E2 -1259.999} C_VEL
LIN {X 0,Y 594.407,Z 167.26,A -85,B 0,C 180,E1 -1262.71,E2 -1262.71} C_VEL
LIN {X 0,Y 594.393,Z 167.26,A -85,B 0,C 180,E1 -1265.427,E2 -1265.427} C_VEL
LIN {X 0,Y 594.397,Z 167.258,A -85,B 0,C 180,E1 -1267.472,E2 -1267.472} C_VEL
LIN {X 0,Y 594.388,Z 167.26,A -85,B 0,C 180,E1 -1270.215,E2 -1270.215} C_VEL
LIN {X 0,Y 594.36,Z 167.266,A -85,B 0,C 180,E1 -1272.982,E2 -1272.982} C_VEL
LIN {X 0,Y 594.36,Z 167.261,A -85,B 0,C 180,E1 -1275.324,E2 -1275.324} C_VEL
LIN {X 0,Y 593.683,Z 167.348,A -85,B 0,C 180,E1 -1275.89,E2 -1275.89} C_VEL
LIN {X 0,Y 590.817,Z 167.708,A -85,B 0,C 180,E1 -1276.808,E2 -1276.808} C_VEL
LIN {X 0,Y 588.408,Z 168.009,A -85,B 0,C 180,E1 -1277.547,E2 -1277.547} C_VEL
LIN {X 0,Y 587.387,Z 168.134,A -85,B 0,C 180,E1 -1278.117,E2 -1278.117} C_VEL
LIN {X 0,Y 587.31,Z 168.142,A -85,B 0,C 180,E1 -1278.31,E2 -1278.31} C_VEL
LIN {X 0,Y 587.332,Z 168.138,A -85,B 0,C 180,E1 -1281.037,E2 -1281.037} C_VEL
LIN {X 0,Y 587.312,Z 168.143,A -85,B 0,C 180,E1 -1283.258,E2 -1283.258} C_VEL
LIN {X 0,Y 587.338,Z 168.138,A -85,B 0,C 180,E1 -1285.516,E2 -1285.516} C_VEL
LIN {X 0,Y 587.348,Z 168.135,A -85,B 0,C 180,E1 -1287.817,E2 -1287.817} C_VEL
LIN {X 0,Y 587.334,Z 168.138,A -85,B 0,C 180,E1 -1290.509,E2 -1290.509} C_VEL
LIN {X 0,Y 587.335,Z 168.141,A -85,B 0,C 180,E1 -1293.396,E2 -1293.396} C_VEL
LIN {X 0,Y 587.346,Z 168.139,A -85,B 0,C 180,E1 -1295.895,E2 -1295.895} C_VEL
LIN {X 0,Y 587.316,Z 168.143,A -85,B 0,C 180,E1 -1298.479,E2 -1298.479} C_VEL
LIN {X 0,Y 587.335,Z 168.14,A -85,B 0,C 180,E1 -1301.156,E2 -1301.156} C_VEL
LIN {X 0,Y 587.322,Z 168.139,A -85,B 0,C 180,E1 -1304.112,E2 -1304.112} C_VEL
LIN {X 0,Y 587.308,Z 168.14,A -85,B 0,C 180,E1 -1306.993,E2 -1306.993} C_VEL
LIN {X 0,Y 587.307,Z 168.142,A -85,B 0,C 180,E1 -1309.745,E2 -1309.745} C_VEL
LIN {X 0,Y 587.34,Z 168.139,A -85,B 0,C 180,E1 -1312.392,E2 -1312.392} C_VEL
LIN {X 0,Y 587.346,Z 168.138,A -85,B 0,C 180,E1 -1314.945,E2 -1314.945} C_VEL
LIN {X 0,Y 587.336,Z 168.138,A -85,B 0,C 180,E1 -1317.421,E2 -1317.421} C_VEL
LIN {X 0,Y 587.342,Z 168.137,A -85,B 0,C 180,E1 -1319.83,E2 -1319.83} C_VEL
LIN {X 0,Y 587.345,Z 168.136,A -85,B 0,C 180,E1 -1322.306,E2 -1322.306} C_VEL
LIN {X 0,Y 587.326,Z 168.138,A -85,B 0,C 180,E1 -1324.483,E2 -1324.483} C_VEL
LIN {X 0,Y 587.313,Z 168.14,A -85,B 0,C 180,E1 -1327.13,E2 -1327.13} C_VEL
LIN {X 0,Y 587.33,Z 168.138,A -85,B 0,C 180,E1 -1329.695,E2 -1329.695} C_VEL
LIN {X 0,Y 587.341,Z 168.136,A -85,B 0,C 180,E1 -1332.594,E2 -1332.594} C_VEL
LIN {X 0,Y 587.356,Z 168.136,A -85,B 0,C 180,E1 -1335.739,E2 -1335.739} C_VEL
LIN {X 0,Y 587.336,Z 168.139,A -85,B 0,C 180,E1 -1338.263,E2 -1338.263} C_VEL
LIN {X 0,Y 587.343,Z 168.137,A -85,B 0,C 180,E1 -1341.051,E2 -1341.051} C_VEL
LIN {X 0,Y 587.311,Z 168.139,A -85,B 0,C 180,E1 -1343.817,E2 -1343.817} C_VEL
LIN {X 0,Y 587.306,Z 168.143,A -85,B 0,C 180,E1 -1345.883,E2 -1345.883} C_VEL
LIN {X 0,Y 587.353,Z 168.135,A -85,B 0,C 180,E1 -1347.943,E2 -1347.943} C_VEL
LIN {X 0,Y 587.385,Z 168.133,A -85,B 0,C 180,E1 -1350.685,E2 -1350.685} C_VEL
LIN {X 0,Y 587.332,Z 168.141,A -85,B 0,C 180,E1 -1353.43,E2 -1353.43} C_VEL
LIN {X 0,Y 587.352,Z 168.135,A -85,B 0,C 180,E1 -1355.493,E2 -1355.493} C_VEL
LIN {X 0,Y 587.36,Z 168.135,A -85,B 0,C 180,E1 -1358.255,E2 -1358.255} C_VEL
LIN {X 0,Y 587.353,Z 168.138,A -85,B 0,C 180,E1 -1361.141,E2 -1361.141} C_VEL
LIN {X 0,Y 587.283,Z 168.144,A -85,B 0,C 180,E1 -1363.142,E2 -1363.142} C_VEL
LIN {X 0,Y 587.246,Z 168.367,A -85,B 0,C 180,E1 -1363.848,E2 -1363.848} C_VEL
LIN {X 0,Y 587.284,Z 173.521,A -85,B 0,C 180,E1 -1366.797,E2 -1366.797} C_VEL
LIN {X 0,Y 587.222,Z 178.469,A -85,B 0,C 180,E1 -1369.579,E2 -1369.579} C_VEL
LIN {X 0,Y 587.215,Z 182.433,A -85,B 0,C 180,E1 -1371.778,E2 -1371.778} C_VEL
LIN {X 0,Y 587.183,Z 187.335,A -85,B 0,C 180,E1 -1374.546,E2 -1374.546} C_VEL
LIN {X 0,Y 587.12,Z 192.038,A -85,B 0,C 180,E1 -1377.057,E2 -1377.057} C_VEL
LIN {X 0,Y 587.146,Z 196.466,A -85,B 0,C 180,E1 -1379.39,E2 -1379.39} C_VEL
LIN {X 0,Y 587.126,Z 201.1,A -85,B 0,C 180,E1 -1381.803,E2 -1381.803} C_VEL
LIN {X 0,Y 587.136,Z 205.979,A -85,B 0,C 180,E1 -1384.319,E2 -1384.319} C_VEL
LIN {X 0,Y 587.145,Z 209.731,A -85,B 0,C 180,E1 -1386.229,E2 -1386.229} C_VEL
LIN {X 0,Y 587.431,Z 217.968,A -85,B 0,C 180,E1 -1386.465,E2 -1386.465} C_VEL
LIN {X 0,Y 587.353,Z 227.752,A -85,B 0,C 180,E1 -1386.854,E2 -1386.854} C_VEL
LIN {X 0,Y 587.34,Z 235.975,A -85,B 0,C 180,E1 -1387.284,E2 -1387.284} C_VEL
LIN {X 0,Y 587.327,Z 244.366,A -85,B 0,C 180,E1 -1387.839,E2 -1387.839} C_VEL
LIN {X 0,Y 587.256,Z 253.303,A -85,B 0,C 180,E1 -1388.597,E2 -1388.597} C_VEL
LIN {X 0,Y 587.25,Z 260.389,A -85,B 0,C 180,E1 -1389.367,E2 -1389.367} C_VEL
LIN {X 0,Y 587.215,Z 265.214,A -85,B 0,C 180,E1 -1390.008,E2 -1390.008} C_VEL
LIN {X 0,Y 587.173,Z 270.413,A -85,B 0,C 180,E1 -1390.86,E2 -1390.86} C_VEL
LIN {X 0,Y 587.166,Z 274.068,A -85,B 0,C 180,E1 -1391.629,E2 -1391.629} C_VEL
LIN {X 0,Y 587.162,Z 277.392,A -85,B 0,C 180,E1 -1392.553,E2 -1392.553} C_VEL
LIN {X 0,Y 587.148,Z 278.765,A -85,B 0,C 180,E1 -1393.102,E2 -1393.102} C_VEL
LIN {X 0,Y 587.149,Z 280.457,A -85,B 0,C 180,E1 -1394.097,E2 -1394.097} C_VEL
LIN {X 0,Y 587.137,Z 280.998,A -85,B 0,C 180,E1 -1395.073,E2 -1395.073} C_VEL
LIN {X 0,Y 587.131,Z 280.403,A -85,B 0,C 180,E1 -1396.033,E2 -1396.033} C_VEL
LIN {X 0,Y 587.161,Z 278.781,A -85,B 0,C 180,E1 -1396.981,E2 -1396.981} C_VEL
LIN {X 0,Y 587.187,Z 276.136,A -85,B 0,C 180,E1 -1397.914,E2 -1397.914} C_VEL
LIN {X 0,Y 587.179,Z 271.938,A -85,B 0,C 180,E1 -1398.943,E2 -1398.943} C_VEL
LIN {X 0,Y 587.208,Z 267.542,A -85,B 0,C 180,E1 -1399.738,E2 -1399.738} C_VEL
LIN {X 0,Y 587.248,Z 261.122,A -85,B 0,C 180,E1 -1400.634,E2 -1400.634} C_VEL
LIN {X 0,Y 587.252,Z 255.267,A -85,B 0,C 180,E1 -1401.294,E2 -1401.294} C_VEL
LIN {X 0,Y 587.273,Z 247.945,A -85,B 0,C 180,E1 -1401.969,E2 -1401.969} C_VEL
LIN {X 0,Y 587.302,Z 239.325,A -85,B 0,C 180,E1 -1402.606,E2 -1402.606} C_VEL
LIN {X 0,Y 587.336,Z 229.686,A -85,B 0,C 180,E1 -1403.146,E2 -1403.146} C_VEL
LIN {X 0,Y 587.397,Z 220.768,A -85,B 0,C 180,E1 -1403.525,E2 -1403.525} C_VEL
LIN {X 0,Y 587.41,Z 212.258,A -85,B 0,C 180,E1 -1403.791,E2 -1403.791} C_VEL
LIN {X 0,Y 587.142,Z 209.676,A -85,B 0,C 180,E1 -1403.879,E2 -1403.879} C_VEL
LIN {X 0,Y 587.139,Z 203.748,A -85,B 0,C 180,E1 -1406.918,E2 -1406.918} C_VEL
LIN {X 0,Y 587.154,Z 198.147,A -85,B 0,C 180,E1 -1409.821,E2 -1409.821} C_VEL
LIN {X 0,Y 587.166,Z 193.342,A -85,B 0,C 180,E1 -1412.342,E2 -1412.342} C_VEL
LIN {X 0,Y 587.173,Z 187.911,A -85,B 0,C 180,E1 -1415.234,E2 -1415.234} C_VEL
LIN {X 0,Y 587.228,Z 183.922,A -85,B 0,C 180,E1 -1417.483,E2 -1417.483} C_VEL
LIN {X 0,Y 587.205,Z 180.096,A -85,B 0,C 180,E1 -1419.692,E2 -1419.692} C_VEL
LIN {X 0,Y 587.236,Z 176.134,A -85,B 0,C 180,E1 -1421.871,E2 -1421.871} C_VEL
LIN {X 0,Y 587.243,Z 172.345,A -85,B 0,C 180,E1 -1424.023,E2 -1424.023} C_VEL
LIN {X 0,Y 587.26,Z 168.557,A -85,B 0,C 180,E1 -1426.153,E2 -1426.153} C_VEL
LIN {X 0,Y 587.289,Z 168.145,A -85,B 0,C 180,E1 -1426.858,E2 -1426.858} C_VEL
LIN {X 0,Y 587.337,Z 168.139,A -85,B 0,C 180,E1 -1428.963,E2 -1428.963} C_VEL
LIN {X 0,Y 587.365,Z 168.135,A -85,B 0,C 180,E1 -1431.745,E2 -1431.745} C_VEL
LIN {X 0,Y 587.358,Z 168.139,A -85,B 0,C 180,E1 -1434.508,E2 -1434.508} C_VEL
LIN {X 0,Y 587.366,Z 168.134,A -85,B 0,C 180,E1 -1437.257,E2 -1437.257} C_VEL
LIN {X 0,Y 587.381,Z 168.133,A -85,B 0,C 180,E1 -1440.001,E2 -1440.001} C_VEL
LIN {X 0,Y 587.375,Z 168.134,A -85,B 0,C 180,E1 -1442.744,E2 -1442.744} C_VEL
LIN {X 0,Y 587.353,Z 168.136,A -85,B 0,C 180,E1 -1445.494,E2 -1445.494} C_VEL
LIN {X 0,Y 587.364,Z 168.134,A -85,B 0,C 180,E1 -1447.564,E2 -1447.564} C_VEL
LIN {X 0,Y 587.343,Z 168.138,A -85,B 0,C 180,E1 -1450.34,E2 -1450.34} C_VEL
LIN {X 0,Y 587.317,Z 168.141,A -85,B 0,C 180,E1 -1453.142,E2 -1453.142} C_VEL
LIN {X 0,Y 587.332,Z 168.14,A -85,B 0,C 180,E1 -1455.264,E2 -1455.264} C_VEL
LIN {X 0,Y 587.349,Z 168.139,A -85,B 0,C 180,E1 -1457.406,E2 -1457.406} C_VEL
LIN {X 0,Y 587.344,Z 168.139,A -85,B 0,C 180,E1 -1459.575,E2 -1459.575} C_VEL
LIN {X 0,Y 587.338,Z 168.137,A -85,B 0,C 180,E1 -1462.514,E2 -1462.514} C_VEL
LIN {X 0,Y 587.339,Z 168.14,A -85,B 0,C 180,E1 -1465.517,E2 -1465.517} C_VEL
LIN {X 0,Y 587.341,Z 168.139,A -85,B 0,C 180,E1 -1467.818,E2 -1467.818} C_VEL
LIN {X 0,Y 587.338,Z 168.137,A -85,B 0,C 180,E1 -1470.51,E2 -1470.51} C_VEL
LIN {X 0,Y 587.338,Z 168.14,A -85,B 0,C 180,E1 -1473.397,E2 -1473.397} C_VEL
LIN {X 0,Y 587.294,Z 168.145,A -85,B 0,C 180,E1 -1475.9,E2 -1475.9} C_VEL
LIN {X 0,Y 587.326,Z 168.139,A -85,B 0,C 180,E1 -1478.48,E2 -1478.48} C_VEL
LIN {X 0,Y 587.337,Z 168.138,A -85,B 0,C 180,E1 -1481.157,E2 -1481.157} C_VEL
LIN {X 0,Y 587.329,Z 168.139,A -85,B 0,C 180,E1 -1484.114,E2 -1484.114} C_VEL
LIN {X 0,Y 587.312,Z 168.142,A -85,B 0,C 180,E1 -1486.993,E2 -1486.993} C_VEL
LIN {X 0,Y 587.313,Z 168.142,A -85,B 0,C 180,E1 -1489.746,E2 -1489.746} C_VEL
LIN {X 0,Y 587.346,Z 168.137,A -85,B 0,C 180,E1 -1492.392,E2 -1492.392} C_VEL
LIN {X 0,Y 587.356,Z 168.137,A -85,B 0,C 180,E1 -1495.651,E2 -1495.651} C_VEL
LIN {X 0,Y 587.363,Z 168.138,A -85,B 0,C 180,E1 -1498.735,E2 -1498.735} C_VEL
LIN {X 0,Y 587.465,Z 168.858,A -85,B 0,C 180,E1 -1499.041,E2 -1499.041} C_VEL
LIN {X 0,Y 587.6,Z 174.835,A -85,B 0,C 180,E1 -1500.823,E2 -1500.823} C_VEL
LIN {X 0,Y 587.429,Z 183.686,A -85,B 0,C 180,E1 -1503.343,E2 -1503.343} C_VEL
LIN {X 0,Y 587.458,Z 193.597,A -85,B 0,C 180,E1 -1505.999,E2 -1505.999} C_VEL
LIN {X 0,Y 587.369,Z 204.635,A -85,B 0,C 180,E1 -1508.964,E2 -1508.964} C_VEL
LIN {X 0,Y 587.326,Z 214.314,A -85,B 0,C 180,E1 -1511.512,E2 -1511.512} C_VEL
LIN {X 0,Y 587.263,Z 225.376,A -85,B 0,C 180,E1 -1514.379,E2 -1514.379} C_VEL
LIN {X 0,Y 587.246,Z 236.438,A -85,B 0,C 180,E1 -1517.209,E2 -1517.209} C_VEL
LIN {X 0,Y 587.208,Z 247.5,A -85,B 0,C 180,E1 -1520.006,E2 -1520.006} C_VEL
LIN {X 0,Y 587.216,Z 248.883,A -85,B 0,C 180,E1 -1520.354,E2 -1520.354} C_VEL
LIN {X 0,Y 587.497,Z 255.587,A -85,B 0,C 180,E1 -1520.511,E2 -1520.511} C_VEL
LIN {X 0,Y 587.465,Z 264.895,A -85,B 0,C 180,E1 -1520.793,E2 -1520.793} C_VEL
LIN {X 0,Y 587.403,Z 273.401,A -85,B 0,C 180,E1 -1521.139,E2 -1521.139} C_VEL
LIN {X 0,Y 587.377,Z 281.73,A -85,B 0,C 180,E1 -1521.572,E2 -1521.572} C_VEL
LIN {X 0,Y 587.346,Z 289.767,A -85,B 0,C 180,E1 -1522.091,E2 -1522.091} C_VEL
LIN {X 0,Y 587.292,Z 297.417,A -85,B 0,C 180,E1 -1522.695,E2 -1522.695} C_VEL
LIN {X 0,Y 587.281,Z 305.812,A -85,B 0,C 180,E1 -1523.513,E2 -1523.513} C_VEL
LIN {X 0,Y 587.239,Z 312.433,A -85,B 0,C 180,E1 -1524.334,E2 -1524.334} C_VEL
LIN {X 0,Y 587.17,Z 317.987,A -85,B 0,C 180,E1 -1525.194,E2 -1525.194} C_VEL
LIN {X 0,Y 587.21,Z 323.148,A -85,B 0,C 180,E1 -1526.226,E2 -1526.226} C_VEL
LIN {X 0,Y 587.155,Z 325.789,A -85,B 0,C 180,E1 -1526.912,E2 -1526.912} C_VEL
LIN {X 0,Y 587.141,Z 328.681,A -85,B 0,C 180,E1 -1527.942,E2 -1527.942} C_VEL
LIN {X 0,Y 587.145,Z 329.936,A -85,B 0,C 180,E1 -1528.628,E2 -1528.628} C_VEL
LIN {X 0,Y 587.136,Z 330.712,A -85,B 0,C 180,E1 -1529.314,E2 -1529.314} C_VEL
LIN {X 0,Y 587.134,Z 331,A -85,B 0,C 180,E1 -1530,E2 -1530} C_VEL
LIN {X 0,Y 587.136,Z 330.711,A -85,B 0,C 180,E1 -1530.686,E2 -1530.686} C_VEL
LIN {X 0,Y 587.145,Z 329.936,A -85,B 0,C 180,E1 -1531.372,E2 -1531.372} C_VEL
LIN {X 0,Y 587.141,Z 328.68,A -85,B 0,C 180,E1 -1532.058,E2 -1532.058} C_VEL
LIN {X 0,Y 587.155,Z 325.787,A -85,B 0,C 180,E1 -1533.088,E2 -1533.088} C_VEL
LIN {X 0,Y 587.21,Z 323.147,A -85,B 0,C 180,E1 -1533.774,E2 -1533.774} C_VEL
LIN {X 0,Y 587.17,Z 317.984,A -85,B 0,C 180,E1 -1534.806,E2 -1534.806} C_VEL
LIN {X 0,Y 587.253,Z 311.187,A -85,B 0,C 180,E1 -1535.839,E2 -1535.839} C_VEL
LIN {X 0,Y 587.269,Z 304.287,A -85,B 0,C 180,E1 -1536.645,E2 -1536.645} C_VEL
LIN {X 0,Y 587.297,Z 296.404,A -85,B 0,C 180,E1 -1537.391,E2 -1537.391} C_VEL
LIN {X 0,Y 587.359,Z 288.547,A -85,B 0,C 180,E1 -1537.996,E2 -1537.996} C_VEL
LIN {X 0,Y 587.403,Z 278.731,A -85,B 0,C 180,E1 -1538.601,E2 -1538.601} C_VEL
LIN {X 0,Y 587.461,Z 267.295,A -85,B 0,C 180,E1 -1539.121,E2 -1539.121} C_VEL
LIN {X 0,Y 587.503,Z 257.239,A -85,B 0,C 180,E1 -1539.446,E2 -1539.446} C_VEL
LIN {X 0,Y 587.27,Z 249.731,A -85,B 0,C 180,E1 -1539.623,E2 -1539.623} C_VEL
LIN {X 0,Y 587.204,Z 248.882,A -85,B 0,C 180,E1 -1539.646,E2 -1539.646} C_VEL
LIN {X 0,Y 587.241,Z 237.82,A -85,B 0,C 180,E1 -1542.44,E2 -1542.44} C_VEL
LIN {X 0,Y 587.274,Z 226.758,A -85,B 0,C 180,E1 -1545.265,E2 -1545.265} C_VEL
LIN {X 0,Y 587.311,Z 215.696,A -85,B 0,C 180,E1 -1548.127,E2 -1548.127} C_VEL
LIN {X 0,Y 587.361,Z 206.016,A -85,B 0,C 180,E1 -1550.67,E2 -1550.67} C_VEL
LIN {X 0,Y 587.411,Z 194.887,A -85,B 0,C 180,E1 -1553.629,E2 -1553.629} C_VEL
LIN {X 0,Y 587.433,Z 185.018,A -85,B 0,C 180,E1 -1556.274,E2 -1556.274} C_VEL
LIN {X 0,Y 587.57,Z 175.919,A -85,B 0,C 180,E1 -1558.881,E2 -1558.881} C_VEL
LIN {X 0,Y 587.618,Z 170.136,A -85,B 0,C 180,E1 -1560.556,E2 -1560.556} C_VEL
LIN {X 0,Y 587.359,Z 168.138,A -85,B 0,C 180,E1 -1561.165,E2 -1561.165} C_VEL
LIN {X 0,Y 587.362,Z 168.136,A -85,B 0,C 180,E1 -1564.22,E2 -1564.22} C_VEL
LIN {X 0,Y 587.347,Z 168.137,A -85,B 0,C 180,E1 -1567.608,E2 -1567.608} C_VEL
LIN {X 0,Y 587.313,Z 168.142,A -85,B 0,C 180,E1 -1570.255,E2 -1570.255} C_VEL
LIN {X 0,Y 587.307,Z 168.143,A -85,B 0,C 180,E1 -1573.117,E2 -1573.117} C_VEL
LIN {X 0,Y 587.316,Z 168.139,A -85,B 0,C 180,E1 -1576.049,E2 -1576.049} C_VEL
LIN {X 0,Y 587.338,Z 168.137,A -85,B 0,C 180,E1 -1578.925,E2 -1578.925} C_VEL
LIN {X 0,Y 587.324,Z 168.139,A -85,B 0,C 180,E1 -1581.52,E2 -1581.52} C_VEL
LIN {X 0,Y 587.291,Z 168.143,A -85,B 0,C 180,E1 -1584.1,E2 -1584.1} C_VEL
LIN {X 0,Y 587.338,Z 168.137,A -85,B 0,C 180,E1 -1586.603,E2 -1586.603} C_VEL
LIN {X 0,Y 587.339,Z 168.14,A -85,B 0,C 180,E1 -1589.491,E2 -1589.491} C_VEL
LIN {X 0,Y 587.345,Z 168.137,A -85,B 0,C 180,E1 -1592.309,E2 -1592.309} C_VEL
LIN {X 0,Y 587.339,Z 168.139,A -85,B 0,C 180,E1 -1594.483,E2 -1594.483} C_VEL
LIN {X 0,Y 587.343,Z 168.137,A -85,B 0,C 180,E1 -1597.486,E2 -1597.486} C_VEL
LIN {X 0,Y 587.326,Z 168.141,A -85,B 0,C 180,E1 -1599.695,E2 -1599.695} C_VEL
LIN {X 0,Y 587.309,Z 168.141,A -85,B 0,C 180,E1 -1601.872,E2 -1601.872} C_VEL
LIN {X 0,Y 587.327,Z 168.138,A -85,B 0,C 180,E1 -1604.024,E2 -1604.024} C_VEL
LIN {X 0,Y 587.36,Z 168.138,A -85,B 0,C 180,E1 -1606.154,E2 -1606.154} C_VEL
LIN {X 0,Y 587.342,Z 168.138,A -85,B 0,C 180,E1 -1608.962,E2 -1608.962} C_VEL
LIN {X 0,Y 587.347,Z 168.136,A -85,B 0,C 180,E1 -1611.744,E2 -1611.744} C_VEL
LIN {X 0,Y 587.347,Z 168.135,A -85,B 0,C 180,E1 -1614.506,E2 -1614.506} C_VEL
LIN {X 0,Y 587.372,Z 168.133,A -85,B 0,C 180,E1 -1617.256,E2 -1617.256} C_VEL
LIN {X 0,Y 587.388,Z 168.132,A -85,B 0,C 180,E1 -1619.999,E2 -1619.999} C_VEL
LIN {X 0,Y 587.374,Z 168.136,A -85,B 0,C 180,E1 -1622.743,E2 -1622.743} C_VEL
LIN {X 0,Y 587.357,Z 168.136,A -85,B 0,C 180,E1 -1625.492,E2 -1625.492} C_VEL
LIN {X 0,Y 587.342,Z 168.137,A -85,B 0,C 180,E1 -1628.255,E2 -1628.255} C_VEL
LIN {X 0,Y 587.352,Z 168.135,A -85,B 0,C 180,E1 -1631.133,E2 -1631.133} C_VEL
LIN {X 0,Y 587.367,Z 168.137,A -85,B 0,C 180,E1 -1634.259,E2 -1634.259} C_VEL
LIN {X 0,Y 587.344,Z 168.136,A -85,B 0,C 180,E1 -1637.405,E2 -1637.405} C_VEL
LIN {X 0,Y 587.31,Z 168.142,A -85,B 0,C 180,E1 -1638.31,E2 -1638.31} C_VEL
LIN {X 0,Y 586.668,Z 168.221,A -85,B 0,C 180,E1 -1638.882,E2 -1638.882} C_VEL
LIN {X 0,Y 583.844,Z 168.572,A -85,B 0,C 180,E1 -1639.81,E2 -1639.81} C_VEL
LIN {X 0,Y 581.433,Z 168.875,A -85,B 0,C 180,E1 -1640.557,E2 -1640.557} C_VEL
LIN {X 0,Y 580.379,Z 169.004,A -85,B 0,C 180,E1 -1641.134,E2 -1641.134} C_VEL
LIN {X 0,Y 580.284,Z 169.015,A -85,B 0,C 180,E1 -1641.329,E2 -1641.329} C_VEL
LIN {X 0,Y 580.296,Z 169.016,A -85,B 0,C 180,E1 -1644.316,E2 -1644.316} C_VEL
LIN {X 0,Y 580.279,Z 169.017,A -85,B 0,C 180,E1 -1646.622,E2 -1646.622} C_VEL
LIN {X 0,Y 580.303,Z 169.014,A -85,B 0,C 180,E1 -1649.309,E2 -1649.309} C_VEL
LIN {X 0,Y 580.298,Z 169.017,A -85,B 0,C 180,E1 -1652.199,E2 -1652.199} C_VEL
LIN {X 0,Y 580.289,Z 169.018,A -85,B 0,C 180,E1 -1654.695,E2 -1654.695} C_VEL
LIN {X 0,Y 580.297,Z 169.017,A -85,B 0,C 180,E1 -1657.267,E2 -1657.267} C_VEL
LIN {X 0,Y 580.298,Z 169.014,A -85,B 0,C 180,E1 -1660.271,E2 -1660.271} C_VEL
LIN {X 0,Y 580.273,Z 169.017,A -85,B 0,C 180,E1 -1662.705,E2 -1662.705} C_VEL
LIN {X 0,Y 580.265,Z 169.018,A -85,B 0,C 180,E1 -1665.608,E2 -1665.608} C_VEL
LIN {X 0,Y 580.309,Z 169.012,A -85,B 0,C 180,E1 -1668.233,E2 -1668.233} C_VEL
LIN {X 0,Y 580.275,Z 169.017,A -85,B 0,C 180,E1 -1670.964,E2 -1670.964} C_VEL
LIN {X 0,Y 580.289,Z 169.016,A -85,B 0,C 180,E1 -1673.598,E2 -1673.598} C_VEL
LIN {X 0,Y 580.317,Z 169.013,A -85,B 0,C 180,E1 -1676.145,E2 -1676.145} C_VEL
LIN {X 0,Y 580.285,Z 169.016,A -85,B 0,C 180,E1 -1678.615,E2 -1678.615} C_VEL
LIN {X 0,Y 580.289,Z 169.015,A -85,B 0,C 180,E1 -1681.023,E2 -1681.023} C_VEL
LIN {X 0,Y 580.285,Z 169.016,A -85,B 0,C 180,E1 -1683.665,E2 -1683.665} C_VEL
LIN {X 0,Y 580.294,Z 169.015,A -85,B 0,C 180,E1 -1685.683,E2 -1685.683} C_VEL
LIN {X 0,Y 580.267,Z 169.02,A -85,B 0,C 180,E1 -1687.947,E2 -1687.947} C_VEL
LIN {X 0,Y 580.31,Z 169.012,A -85,B 0,C 180,E1 -1690.914,E2 -1690.914} C_VEL
LIN {X 0,Y 580.276,Z 169.017,A -85,B 0,C 180,E1 -1693.825,E2 -1693.825} C_VEL
LIN {X 0,Y 580.274,Z 169.019,A -85,B 0,C 180,E1 -1696.696,E2 -1696.696} C_VEL
LIN {X 0,Y 580.292,Z 169.016,A -85,B 0,C 180,E1 -1699.533,E2 -1699.533} C_VEL
LIN {X 0,Y 580.311,Z 169.012,A -85,B 0,C 180,E1 -1702.344,E2 -1702.344} C_VEL
LIN {X 0,Y 580.335,Z 169.009,A -85,B 0,C 180,E1 -1705.137,E2 -1705.137} C_VEL
LIN {X 0,Y 580.324,Z 169.011,A -85,B 0,C 180,E1 -1707.918,E2 -1707.918} C_VEL
LIN {X 0,Y 580.355,Z 169.009,A -85,B 0,C 180,E1 -1710.694,E2 -1710.694} C_VEL
LIN {X 0,Y 580.283,Z 169.019,A -85,B 0,C 180,E1 -1713.472,E2 -1713.472} C_VEL
LIN {X 0,Y 580.318,Z 169.011,A -85,B 0,C 180,E1 -1715.56,E2 -1715.56} C_VEL
LIN {X 0,Y 580.325,Z 169.012,A -85,B 0,C 180,E1 -1718.356,E2 -1718.356} C_VEL
LIN {X 0,Y 580.325,Z 169.013,A -85,B 0,C 180,E1 -1721.208,E2 -1721.208} C_VEL
LIN {X 0,Y 580.215,Z 169.025,A -85,B 0,C 180,E1 -1723.305,E2 -1723.305} C_VEL
LIN {X 0,Y 580.194,Z 169.41,A -85,B 0,C 180,E1 -1724.02,E2 -1724.02} C_VEL
LIN {X 0,Y 580.213,Z 174.406,A -85,B 0,C 180,E1 -1726.9,E2 -1726.9} C_VEL
LIN {X 0,Y 580.159,Z 179.554,A -85,B 0,C 180,E1 -1729.827,E2 -1729.827} C_VEL
LIN {X 0,Y 580.163,Z 184.883,A -85,B 0,C 180,E1 -1732.808,E2 -1732.808} C_VEL
LIN {X 0,Y 580.062,Z 188.893,A -85,B 0,C 180,E1 -1735.091,E2 -1735.091} C_VEL
LIN {X 0,Y 580.034,Z 193.13,A -85,B 0,C 180,E1 -1737.415,E2 -1737.415} C_VEL
LIN {X 0,Y 580.052,Z 197.583,A -85,B 0,C 180,E1 -1739.786,E2 -1739.786} C_VEL
LIN {X 0,Y 580.037,Z 202.203,A -85,B 0,C 180,E1 -1742.217,E2 -1742.217} C_VEL
LIN {X 0,Y 580.037,Z 206.994,A -85,B 0,C 180,E1 -1744.713,E2 -1744.713} C_VEL
LIN {X 0,Y 580.051,Z 209.703,A -85,B 0,C 180,E1 -1746.117,E2 -1746.117} C_VEL
LIN {X 0,Y 580.427,Z 216.181,A -85,B 0,C 180,E1 -1746.299,E2 -1746.299} C_VEL
LIN {X 0,Y 580.347,Z 226.377,A -85,B 0,C 180,E1 -1746.69,E2 -1746.69} C_VEL
LIN {X 0,Y 580.315,Z 233.992,A -85,B 0,C 180,E1 -1747.074,E2 -1747.074} C_VEL
LIN {X 0,Y 580.267,Z 242.25,A -85,B 0,C 180,E1 -1747.598,E2 -1747.598} C_VEL
LIN {X 0,Y 580.225,Z 249.282,A -85,B 0,C 180,E1 -1748.151,E2 -1748.151} C_VEL
LIN {X 0,Y 580.168,Z 257.334,A -85,B 0,C 180,E1 -1748.932,E2 -1748.932} C_VEL
LIN {X 0,Y 580.164,Z 263.798,A -85,B 0,C 180,E1 -1749.737,E2 -1749.737} C_VEL
LIN {X 0,Y 580.105,Z 268.887,A -85,B 0,C 180,E1 -1750.532,E2 -1750.532} C_VEL
LIN {X 0,Y 580.074,Z 272.86,A -85,B 0,C 180,E1 -1751.31,E2 -1751.31} C_VEL
LIN {X 0,Y 580.097,Z 274.916,A -85,B 0,C 180,E1 -1751.785,E2 -1751.785} C_VEL
LIN {X 0,Y 580.072,Z 277.944,A -85,B 0,C 180,E1 -1752.725,E2 -1752.725} C_VEL
LIN {X 0,Y 580.023,Z 279.908,A -85,B 0,C 180,E1 -1753.682,E2 -1753.682} C_VEL
LIN {X 0,Y 580.028,Z 280.847,A -85,B 0,C 180,E1 -1754.649,E2 -1754.649} C_VEL
LIN {X 0,Y 580.033,Z 280.759,A -85,B 0,C 180,E1 -1755.633,E2 -1755.633} C_VEL
LIN {X 0,Y 580.028,Z 279.584,A -85,B 0,C 180,E1 -1756.635,E2 -1756.635} C_VEL
LIN {X 0,Y 580.08,Z 277.122,A -85,B 0,C 180,E1 -1757.65,E2 -1757.65} C_VEL
LIN {X 0,Y 580.085,Z 274.18,A -85,B 0,C 180,E1 -1758.478,E2 -1758.478} C_VEL
LIN {X 0,Y 580.104,Z 269.376,A -85,B 0,C 180,E1 -1759.47,E2 -1759.47} C_VEL
LIN {X 0,Y 580.159,Z 262.973,A -85,B 0,C 180,E1 -1760.471,E2 -1760.471} C_VEL
LIN {X 0,Y 580.19,Z 254.936,A -85,B 0,C 180,E1 -1761.405,E2 -1761.405} C_VEL
LIN {X 0,Y 580.224,Z 247.239,A -85,B 0,C 180,E1 -1762.114,E2 -1762.114} C_VEL
LIN {X 0,Y 580.261,Z 237.207,A -85,B 0,C 180,E1 -1762.829,E2 -1762.829} C_VEL
LIN {X 0,Y 580.31,Z 228.296,A -85,B 0,C 180,E1 -1763.311,E2 -1763.311} C_VEL
LIN {X 0,Y 580.389,Z 220.08,A -85,B 0,C 180,E1 -1763.653,E2 -1763.653} C_VEL
LIN {X 0,Y 580.309,Z 212.13,A -85,B 0,C 180,E1 -1763.903,E2 -1763.903} C_VEL
LIN {X 0,Y 580.062,Z 209.69,A -85,B 0,C 180,E1 -1763.98,E2 -1763.98} C_VEL
LIN {X 0,Y 580.063,Z 203.946,A -85,B 0,C 180,E1 -1766.962,E2 -1766.962} C_VEL
LIN {X 0,Y 580.07,Z 199.27,A -85,B 0,C 180,E1 -1769.413,E2 -1769.413} C_VEL
LIN {X 0,Y 580.07,Z 194.046,A -85,B 0,C 180,E1 -1772.184,E2 -1772.184} C_VEL
LIN {X 0,Y 580.074,Z 190.423,A -85,B 0,C 180,E1 -1774.141,E2 -1774.141} C_VEL
LIN {X 0,Y 580.166,Z 185.411,A -85,B 0,C 180,E1 -1777.021,E2 -1777.021} C_VEL
LIN {X 0,Y 580.158,Z 181.218,A -85,B 0,C 180,E1 -1779.434,E2 -1779.434} C_VEL
LIN {X 0,Y 580.164,Z 177.245,A -85,B 0,C 180,E1 -1781.642,E2 -1781.642} C_VEL
LIN {X 0,Y 580.206,Z 173.398,A -85,B 0,C 180,E1 -1783.824,E2 -1783.824} C_VEL
LIN {X 0,Y 580.199,Z 169.62,A -85,B 0,C 180,E1 -1785.981,E2 -1785.981} C_VEL
LIN {X 0,Y 580.218,Z 169.027,A -85,B 0,C 180,E1 -1786.695,E2 -1786.695} C_VEL
LIN {X 0,Y 580.306,Z 169.016,A -85,B 0,C 180,E1 -1788.828,E2 -1788.828} C_VEL
LIN {X 0,Y 580.328,Z 169.011,A -85,B 0,C 180,E1 -1791.645,E2 -1791.645} C_VEL
LIN {X 0,Y 580.323,Z 169.015,A -85,B 0,C 180,E1 -1794.441,E2 -1794.441} C_VEL
LIN {X 0,Y 580.334,Z 169.01,A -85,B 0,C 180,E1 -1797.224,E2 -1797.224} C_VEL
LIN {X 0,Y 580.351,Z 169.009,A -85,B 0,C 180,E1 -1800.001,E2 -1800.001} C_VEL
LIN {X 0,Y 580.341,Z 169.01,A -85,B 0,C 180,E1 -1802.777,E2 -1802.777} C_VEL
LIN {X 0,Y 580.321,Z 169.012,A -85,B 0,C 180,E1 -1805.56,E2 -1805.56} C_VEL
LIN {X 0,Y 580.325,Z 169.011,A -85,B 0,C 180,E1 -1807.656,E2 -1807.656} C_VEL
LIN {X 0,Y 580.302,Z 169.017,A -85,B 0,C 180,E1 -1810.467,E2 -1810.467} C_VEL
LIN {X 0,Y 580.274,Z 169.017,A -85,B 0,C 180,E1 -1813.305,E2 -1813.305} C_VEL
LIN {X 0,Y 580.297,Z 169.015,A -85,B 0,C 180,E1 -1815.453,E2 -1815.453} C_VEL
LIN {X 0,Y 580.295,Z 169.016,A -85,B 0,C 180,E1 -1817.625,E2 -1817.625} C_VEL
LIN {X 0,Y 580.306,Z 169.015,A -85,B 0,C 180,E1 -1819.823,E2 -1819.823} C_VEL
LIN {X 0,Y 580.294,Z 169.015,A -85,B 0,C 180,E1 -1822.803,E2 -1822.803} C_VEL
LIN {X 0,Y 580.31,Z 169.013,A -85,B 0,C 180,E1 -1825.08,E2 -1825.08} C_VEL
LIN {X 0,Y 580.297,Z 169.014,A -85,B 0,C 180,E1 -1828.186,E2 -1828.186} C_VEL
LIN {X 0,Y 580.287,Z 169.016,A -85,B 0,C 180,E1 -1830.695,E2 -1830.695} C_VEL
LIN {X 0,Y 580.306,Z 169.015,A -85,B 0,C 180,E1 -1833.317,E2 -1833.317} C_VEL
LIN {X 0,Y 580.25,Z 169.023,A -85,B 0,C 180,E1 -1835.757,E2 -1835.757} C_VEL
LIN {X 0,Y 580.289,Z 169.018,A -85,B 0,C 180,E1 -1838.147,E2 -1838.147} C_VEL
LIN {X 0,Y 580.299,Z 169.014,A -85,B 0,C 180,E1 -1840.844,E2 -1840.844} C_VEL
LIN {X 0,Y 580.281,Z 169.019,A -85,B 0,C 180,E1 -1843.658,E2 -1843.658} C_VEL
LIN {X 0,Y 580.277,Z 169.017,A -85,B 0,C 180,E1 -1846.61,E2 -1846.61} C_VEL
LIN {X 0,Y 580.299,Z 169.015,A -85,B 0,C 180,E1 -1849.157,E2 -1849.157} C_VEL
LIN {X 0,Y 580.292,Z 169.017,A -85,B 0,C 180,E1 -1851.927,E2 -1851.927} C_VEL
LIN {X 0,Y 580.284,Z 169.018,A -85,B 0,C 180,E1 -1854.455,E2 -1854.455} C_VEL
LIN {X 0,Y 580.294,Z 169.017,A -85,B 0,C 180,E1 -1856.975,E2 -1856.975} C_VEL
LIN {X 0,Y 580.301,Z 169.066,A -85,B 0,C 180,E1 -1858.664,E2 -1858.664} C_VEL
LIN {X 0,Y 580.612,Z 172.906,A -85,B 0,C 180,E1 -1859.845,E2 -1859.845} C_VEL
LIN {X 0,Y 580.554,Z 180.494,A -85,B 0,C 180,E1 -1862.094,E2 -1862.094} C_VEL
LIN {X 0,Y 580.394,Z 190.6,A -85,B 0,C 180,E1 -1864.924,E2 -1864.924} C_VEL
LIN {X 0,Y 580.351,Z 199.083,A -85,B 0,C 180,E1 -1867.2,E2 -1867.2} C_VEL
LIN {X 0,Y 580.31,Z 208.783,A -85,B 0,C 180,E1 -1869.809,E2 -1869.809} C_VEL
LIN {X 0,Y 580.259,Z 219.845,A -85,B 0,C 180,E1 -1872.738,E2 -1872.738} C_VEL
LIN {X 0,Y 580.199,Z 231.236,A -85,B 0,C 180,E1 -1875.707,E2 -1875.707} C_VEL
LIN {X 0,Y 580.174,Z 241.969,A -85,B 0,C 180,E1 -1878.47,E2 -1878.47} C_VEL
LIN {X 0,Y 580.152,Z 248.883,A -85,B 0,C 180,E1 -1880.236,E2 -1880.236} C_VEL
LIN {X 0,Y 580.492,Z 255.586,A -85,B 0,C 180,E1 -1880.395,E2 -1880.395} C_VEL
LIN {X 0,Y 580.467,Z 264.894,A -85,B 0,C 180,E1 -1880.681,E2 -1880.681} C_VEL
LIN {X 0,Y 580.392,Z 273.402,A -85,B 0,C 180,E1 -1881.031,E2 -1881.031} C_VEL
LIN {X 0,Y 580.341,Z 281.733,A -85,B 0,C 180,E1 -1881.469,E2 -1881.469} C_VEL
LIN {X 0,Y 580.299,Z 289.769,A -85,B 0,C 180,E1 -1881.994,E2 -1881.994} C_VEL
LIN {X 0,Y 580.241,Z 297.418,A -85,B 0,C 180,E1 -1882.606,E2 -1882.606} C_VEL
LIN {X 0,Y 580.207,Z 305.768,A -85,B 0,C 180,E1 -1883.428,E2 -1883.428} C_VEL
LIN {X 0,Y 580.173,Z 312.434,A -85,B 0,C 180,E1 -1884.265,E2 -1884.265} C_VEL
LIN {X 0,Y 580.084,Z 317.988,A -85,B 0,C 180,E1 -1885.135,E2 -1885.135} C_VEL
LIN {X 0,Y 580.122,Z 323.148,A -85,B 0,C 180,E1 -1886.18,E2 -1886.18} C_VEL
LIN {X 0,Y 580.07,Z 325.789,A -85,B 0,C 180,E1 -1886.875,E2 -1886.875} C_VEL
LIN {X 0,Y 580.04,Z 328.681,A -85,B 0,C 180,E1 -1887.917,E2 -1887.917} C_VEL
LIN {X 0,Y 580.045,Z 329.936,A -85,B 0,C 180,E1 -1888.612,E2 -1888.612} C_VEL
LIN {X 0,Y 580.036,Z 330.711,A -85,B 0,C 180,E1 -1889.306,E2 -1889.306} C_VEL
LIN {X 0,Y 580.034,Z 331,A -85,B 0,C 180,E1 -1890,E2 -1890} C_VEL
LIN {X 0,Y 580.036,Z 330.71,A -85,B 0,C 180,E1 -1890.694,E2 -1890.694} C_VEL
LIN {X 0,Y 580.045,Z 329.935,A -85,B 0,C 180,E1 -1891.389,E2 -1891.389} C_VEL
LIN {X 0,Y 580.04,Z 328.68,A -85,B 0,C 180,E1 -1892.083,E2 -1892.083} C_VEL
LIN {X 0,Y 580.07,Z 325.788,A -85,B 0,C 180,E1 -1893.126,E2 -1893.126} C_VEL
LIN {X 0,Y 580.122,Z 323.147,A -85,B 0,C 180,E1 -1893.821,E2 -1893.821} C_VEL
LIN {X 0,Y 580.084,Z 317.985,A -85,B 0,C 180,E1 -1894.865,E2 -1894.865} C_VEL
LIN {X 0,Y 580.193,Z 311.186,A -85,B 0,C 180,E1 -1895.91,E2 -1895.91} C_VEL
LIN {X 0,Y 580.226,Z 303.496,A -85,B 0,C 180,E1 -1896.808,E2 -1896.808} C_VEL
LIN {X 0,Y 580.254,Z 296.405,A -85,B 0,C 180,E1 -1897.481,E2 -1897.481} C_VEL
LIN {X 0,Y 580.319,Z 288.544,A -85,B 0,C 180,E1 -1898.093,E2 -1898.093} C_VEL
LIN {X 0,Y 580.389,Z 278.729,A -85,B 0,C 180,E1 -1898.706,E2 -1898.706} C_VEL
LIN {X 0,Y 580.453,Z 267.297,A -85,B 0,C 180,E1 -1899.232,E2 -1899.232} C_VEL
LIN {X 0,Y 580.523,Z 257.24,A -85,B 0,C 180,E1 -1899.56,E2 -1899.56} C_VEL
LIN {X 0,Y 580.281,Z 250.378,A -85,B 0,C 180,E1 -1899.729,E2 -1899.729} C_VEL
LIN {X 0,Y 580.141,Z 248.882,A -85,B 0,C 180,E1 -1899.765,E2 -1899.765} C_VEL
LIN {X 0,Y 580.178,Z 237.82,A -85,B 0,C 180,E1 -1902.594,E2 -1902.594} C_VEL
LIN {X 0,Y 580.201,Z 226.758,A -85,B 0,C 180,E1 -1905.456,E2 -1905.456} C_VEL
LIN {X 0,Y 580.264,Z 215.696,A -85,B 0,C 180,E1 -1908.355,E2 -1908.355} C_VEL
LIN {X 0,Y 580.338,Z 206.253,A -85,B 0,C 180,E1 -1910.868,E2 -1910.868} C_VEL
LIN {X 0,Y 580.389,Z 194.733,A -85,B 0,C 180,E1 -1913.932,E2 -1913.932} C_VEL
LIN {X 0,Y 580.452,Z 185.019,A -85,B 0,C 180,E1 -1916.615,E2 -1916.615} C_VEL
LIN {X 0,Y 580.622,Z 175.561,A -85,B 0,C 180,E1 -1919.366,E2 -1919.366} C_VEL
LIN {X 0,Y 580.46,Z 169.982,A -85,B 0,C 180,E1 -1921.022,E2 -1921.022} C_VEL
LIN {X 0,Y 580.287,Z 169.019,A -85,B 0,C 180,E1 -1921.385,E2 -1921.385} C_VEL
LIN {X 0,Y 580.317,Z 169.014,A -85,B 0,C 180,E1 -1923.855,E2 -1923.855} C_VEL
LIN {X 0,Y 580.301,Z 169.013,A -85,B 0,C 180,E1 -1927.269,E2 -1927.269} C_VEL
LIN {X 0,Y 580.292,Z 169.017,A -85,B 0,C 180,E1 -1930.27,E2 -1930.27} C_VEL
LIN {X 0,Y 580.275,Z 169.018,A -85,B 0,C 180,E1 -1932.707,E2 -1932.707} C_VEL
LIN {X 0,Y 580.261,Z 169.021,A -85,B 0,C 180,E1 -1935.61,E2 -1935.61} C_VEL
LIN {X 0,Y 580.278,Z 169.018,A -85,B 0,C 180,E1 -1938.231,E2 -1938.231} C_VEL
LIN {X 0,Y 580.272,Z 169.017,A -85,B 0,C 180,E1 -1940.964,E2 -1940.964} C_VEL
LIN {X 0,Y 580.27,Z 169.017,A -85,B 0,C 180,E1 -1943.596,E2 -1943.596} C_VEL
LIN {X 0,Y 580.317,Z 169.012,A -85,B 0,C 180,E1 -1946.145,E2 -1946.145} C_VEL
LIN {X 0,Y 580.274,Z 169.017,A -85,B 0,C 180,E1 -1948.614,E2 -1948.614} C_VEL
LIN {X 0,Y 580.291,Z 169.017,A -85,B 0,C 180,E1 -1951.023,E2 -1951.023} C_VEL
LIN {X 0,Y 580.296,Z 169.015,A -85,B 0,C 180,E1 -1953.666,E2 -1953.666} C_VEL
LIN {X 0,Y 580.297,Z 169.015,A -85,B 0,C 180,E1 -1955.683,E2 -1955.683} C_VEL
LIN {X 0,Y 580.274,Z 169.017,A -85,B 0,C 180,E1 -1957.947,E2 -1957.947} C_VEL
LIN {X 0,Y 580.301,Z 169.016,A -85,B 0,C 180,E1 -1960.913,E2 -1960.913} C_VEL
LIN {X 0,Y 580.277,Z 169.018,A -85,B 0,C 180,E1 -1963.825,E2 -1963.825} C_VEL
LIN {X 0,Y 580.329,Z 169.012,A -85,B 0,C 180,E1 -1965.983,E2 -1965.983} C_VEL
LIN {X 0,Y 580.311,Z 169.015,A -85,B 0,C 180,E1 -1968.827,E2 -1968.827} C_VEL
LIN {X 0,Y 580.315,Z 169.012,A -85,B 0,C 180,E1 -1971.643,E2 -1971.643} C_VEL
LIN {X 0,Y 580.276,Z 169.02,A -85,B 0,C 180,E1 -1973.742,E2 -1973.742} C_VEL
LIN {X 0,Y 580.274,Z 169.017,A -85,B 0,C 180,E1 -1975.832,E2 -1975.832} C_VEL
LIN {X 0,Y 580.328,Z 169.011,A -85,B 0,C 180,E1 -1977.917,E2 -1977.917} C_VEL
LIN {X 0,Y 580.354,Z 169.007,A -85,B 0,C 180,E1 -1980.693,E2 -1980.693} C_VEL
LIN {X 0,Y 580.287,Z 169.015,A -85,B 0,C 180,E1 -1983.471,E2 -1983.471} C_VEL
LIN {X 0,Y 580.323,Z 169.012,A -85,B 0,C 180,E1 -1985.559,E2 -1985.559} C_VEL
LIN {X 0,Y 580.327,Z 169.012,A -85,B 0,C 180,E1 -1987.655,E2 -1987.655} C_VEL
LIN {X 0,Y 580.3,Z 169.017,A -85,B 0,C 180,E1 -1990.466,E2 -1990.466} C_VEL
LIN {X 0,Y 580.301,Z 169.014,A -85,B 0,C 180,E1 -1992.591,E2 -1992.591} C_VEL
LIN {X 0,Y 580.289,Z 169.015,A -85,B 0,C 180,E1 -1994.733,E2 -1994.733} C_VEL
LIN {X 0,Y 580.291,Z 169.015,A -85,B 0,C 180,E1 -1997.624,E2 -1997.624} C_VEL
LIN {X 0,Y 580.288,Z 169.015,A -85,B 0,C 180,E1 -1999.822,E2 -1999.822} C_VEL
LIN {X 0,Y 580.284,Z 169.015,A -85,B 0,C 180,E1 -2001.329,E2 -2001.329} C_VEL
LIN {X 0,Y 579.584,Z 169.106,A -85,B 0,C 180,E1 -2001.908,E2 -2001.908} C_VEL
LIN {X 0,Y 576.704,Z 169.462,A -85,B 0,C 180,E1 -2002.848,E2 -2002.848} C_VEL
LIN {X 0,Y 574.309,Z 169.76,A -85,B 0,C 180,E1 -2003.604,E2 -2003.604} C_VEL
LIN {X 0,Y 573.313,Z 169.885,A -85,B 0,C 180,E1 -2004.188,E2 -2004.188} C_VEL
LIN {X 0,Y 573.248,Z 169.892,A -85,B 0,C 180,E1 -2004.385,E2 -2004.385} C_VEL
LIN {X 0,Y 573.252,Z 169.895,A -85,B 0,C 180,E1 -2006.975,E2 -2006.975} C_VEL
LIN {X 0,Y 573.248,Z 169.895,A -85,B 0,C 180,E1 -2009.488,E2 -2009.488} C_VEL
LIN {X 0,Y 573.254,Z 169.891,A -85,B 0,C 180,E1 -2012.644,E2 -2012.644} C_VEL
LIN {X 0,Y 573.252,Z 169.891,A -85,B 0,C 180,E1 -2015.184,E2 -2015.184} C_VEL
LIN {X 0,Y 573.231,Z 169.894,A -85,B 0,C 180,E1 -2017.807,E2 -2017.807} C_VEL
LIN {X 0,Y 573.267,Z 169.89,A -85,B 0,C 180,E1 -2020.527,E2 -2020.527} C_VEL
LIN {X 0,Y 573.24,Z 169.896,A -85,B 0,C 180,E1 -2023.668,E2 -2023.668} C_VEL
LIN {X 0,Y 573.234,Z 169.893,A -85,B 0,C 180,E1 -2026.64,E2 -2026.64} C_VEL
LIN {X 0,Y 573.239,Z 169.893,A -85,B 0,C 180,E1 -2029.474,E2 -2029.474} C_VEL
LIN {X 0,Y 573.231,Z 169.895,A -85,B 0,C 180,E1 -2032.192,E2 -2032.192} C_VEL
LIN {X 0,Y 573.263,Z 169.891,A -85,B 0,C 180,E1 -2034.816,E2 -2034.816} C_VEL
LIN {X 0,Y 573.251,Z 169.892,A -85,B 0,C 180,E1 -2037.355,E2 -2037.355} C_VEL
LIN {X 0,Y 573.251,Z 169.892,A -85,B 0,C 180,E1 -2039.824,E2 -2039.824} C_VEL
LIN {X 0,Y 573.282,Z 169.887,A -85,B 0,C 180,E1 -2042.234,E2 -2042.234} C_VEL
LIN {X 0,Y 573.267,Z 169.893,A -85,B 0,C 180,E1 -2045.366,E2 -2045.366} C_VEL
LIN {X 0,Y 573.224,Z 169.894,A -85,B 0,C 180,E1 -2048.419,E2 -2048.419} C_VEL
LIN {X 0,Y 573.272,Z 169.89,A -85,B 0,C 180,E1 -2050.727,E2 -2050.727} C_VEL
LIN {X 0,Y 573.252,Z 169.891,A -85,B 0,C 180,E1 -2053.622,E2 -2053.622} C_VEL
LIN {X 0,Y 573.231,Z 169.895,A -85,B 0,C 180,E1 -2056.529,E2 -2056.529} C_VEL
LIN {X 0,Y 573.253,Z 169.891,A -85,B 0,C 180,E1 -2058.745,E2 -2058.745} C_VEL
LIN {X 0,Y 573.301,Z 169.886,A -85,B 0,C 180,E1 -2061.541,E2 -2061.541} C_VEL
LIN {X 0,Y 573.284,Z 169.89,A -85,B 0,C 180,E1 -2064.372,E2 -2064.372} C_VEL
LIN {X 0,Y 573.296,Z 169.886,A -85,B 0,C 180,E1 -2067.892,E2 -2067.892} C_VEL
LIN {X 0,Y 573.325,Z 169.884,A -85,B 0,C 180,E1 -2070.702,E2 -2070.702} C_VEL
LIN {X 0,Y 573.234,Z 169.896,A -85,B 0,C 180,E1 -2073.514,E2 -2073.514} C_VEL
LIN {X 0,Y 573.286,Z 169.888,A -85,B 0,C 180,E1 -2075.628,E2 -2075.628} C_VEL
LIN {X 0,Y 573.281,Z 169.891,A -85,B 0,C 180,E1 -2078.459,E2 -2078.459} C_VEL
LIN {X 0,Y 573.29,Z 169.888,A -85,B 0,C 180,E1 -2081.312,E2 -2081.312} C_VEL
LIN {X 0,Y 573.156,Z 169.905,A -85,B 0,C 180,E1 -2083.472,E2 -2083.472} C_VEL
LIN {X 0,Y 573.142,Z 170.76,A -85,B 0,C 180,E1 -2084.374,E2 -2084.374} C_VEL
LIN {X 0,Y 573.135,Z 175.479,A -85,B 0,C 180,E1 -2087.115,E2 -2087.115} C_VEL
LIN {X 0,Y 573.092,Z 180.641,A -85,B 0,C 180,E1 -2090.082,E2 -2090.082} C_VEL
LIN {X 0,Y 573.079,Z 184.672,A -85,B 0,C 180,E1 -2092.344,E2 -2092.344} C_VEL
LIN {X 0,Y 573.007,Z 189.03,A -85,B 0,C 180,E1 -2094.824,E2 -2094.824} C_VEL
LIN {X 0,Y 572.973,Z 192.846,A -85,B 0,C 180,E1 -2096.99,E2 -2096.99} C_VEL
LIN {X 0,Y 572.97,Z 197.301,A -85,B 0,C 180,E1 -2099.441,E2 -2099.441} C_VEL
LIN {X 0,Y 572.951,Z 202.443,A -85,B 0,C 180,E1 -2102.182,E2 -2102.182} C_VEL
LIN {X 0,Y 572.957,Z 207.277,A -85,B 0,C 180,E1 -2104.733,E2 -2104.733} C_VEL
LIN {X 0,Y 572.965,Z 209.691,A -85,B 0,C 180,E1 -2105.999,E2 -2105.999} C_VEL
LIN {X 0,Y 573.431,Z 216.411,A -85,B 0,C 180,E1 -2106.199,E2 -2106.199} C_VEL
LIN {X 0,Y 573.329,Z 226.4,A -85,B 0,C 180,E1 -2106.588,E2 -2106.588} C_VEL
LIN {X 0,Y 573.284,Z 235.164,A -85,B 0,C 180,E1 -2107.045,E2 -2107.045} C_VEL
LIN {X 0,Y 573.21,Z 242.826,A -85,B 0,C 180,E1 -2107.548,E2 -2107.548} C_VEL
LIN {X 0,Y 573.142,Z 250.739,A -85,B 0,C 180,E1 -2108.193,E2 -2108.193} C_VEL
LIN {X 0,Y 573.101,Z 258.06,A -85,B 0,C 180,E1 -2108.938,E2 -2108.938} C_VEL
LIN {X 0,Y 573.076,Z 264.924,A -85,B 0,C 180,E1 -2109.84,E2 -2109.84} C_VEL
LIN {X 0,Y 573.034,Z 269.252,A -85,B 0,C 180,E1 -2110.543,E2 -2110.543} C_VEL
LIN {X 0,Y 572.996,Z 272.775,A -85,B 0,C 180,E1 -2111.244,E2 -2111.244} C_VEL
LIN {X 0,Y 573.005,Z 275.691,A -85,B 0,C 180,E1 -2111.969,E2 -2111.969} C_VEL
LIN {X 0,Y 572.974,Z 277.745,A -85,B 0,C 180,E1 -2112.614,E2 -2112.614} C_VEL
LIN {X 0,Y 572.924,Z 279.867,A -85,B 0,C 180,E1 -2113.637,E2 -2113.637} C_VEL
LIN {X 0,Y 572.929,Z 280.848,A -85,B 0,C 180,E1 -2114.647,E2 -2114.647} C_VEL
LIN {X 0,Y 572.933,Z 280.759,A -85,B 0,C 180,E1 -2115.638,E2 -2115.638} C_VEL
LIN {X 0,Y 572.93,Z 279.648,A -85,B 0,C 180,E1 -2116.613,E2 -2116.613} C_VEL
LIN {X 0,Y 573.001,Z 277.455,A -85,B 0,C 180,E1 -2117.579,E2 -2117.579} C_VEL
LIN {X 0,Y 573.01,Z 274.16,A -85,B 0,C 180,E1 -2118.525,E2 -2118.525} C_VEL
LIN {X 0,Y 573.01,Z 269.496,A -85,B 0,C 180,E1 -2119.502,E2 -2119.502} C_VEL
LIN {X 0,Y 573.062,Z 264.071,A -85,B 0,C 180,E1 -2120.379,E2 -2120.379} C_VEL
LIN {X 0,Y 573.114,Z 256.801,A -85,B 0,C 180,E1 -2121.289,E2 -2121.289} C_VEL
LIN {X 0,Y 573.147,Z 250.212,A -85,B 0,C 180,E1 -2121.943,E2 -2121.943} C_VEL
LIN {X 0,Y 573.157,Z 242.845,A -85,B 0,C 180,E1 -2122.541,E2 -2122.541} C_VEL
LIN {X 0,Y 573.255,Z 234.603,A -85,B 0,C 180,E1 -2123.079,E2 -2123.079} C_VEL
LIN {X 0,Y 573.354,Z 224.765,A -85,B 0,C 180,E1 -2123.579,E2 -2123.579} C_VEL
LIN {X 0,Y 573.423,Z 213.816,A -85,B 0,C 180,E1 -2123.965,E2 -2123.965} C_VEL
LIN {X 0,Y 572.952,Z 209.669,A -85,B 0,C 180,E1 -2124.103,E2 -2124.103} C_VEL
LIN {X 0,Y 572.962,Z 205.064,A -85,B 0,C 180,E1 -2126.522,E2 -2126.522} C_VEL
LIN {X 0,Y 572.974,Z 200.084,A -85,B 0,C 180,E1 -2129.161,E2 -2129.161} C_VEL
LIN {X 0,Y 572.994,Z 194.778,A -85,B 0,C 180,E1 -2132.02,E2 -2132.02} C_VEL
LIN {X 0,Y 573.019,Z 190.291,A -85,B 0,C 180,E1 -2134.58,E2 -2134.58} C_VEL
LIN {X 0,Y 573.086,Z 185.03,A -85,B 0,C 180,E1 -2137.657,E2 -2137.657} C_VEL
LIN {X 0,Y 573.087,Z 181.001,A -85,B 0,C 180,E1 -2139.918,E2 -2139.918} C_VEL
LIN {X 0,Y 573.141,Z 175.782,A -85,B 0,C 180,E1 -2142.886,E2 -2142.886} C_VEL
LIN {X 0,Y 573.144,Z 170.706,A -85,B 0,C 180,E1 -2145.805,E2 -2145.805} C_VEL
LIN {X 0,Y 573.16,Z 169.908,A -85,B 0,C 180,E1 -2146.528,E2 -2146.528} C_VEL
LIN {X 0,Y 573.264,Z 169.894,A -85,B 0,C 180,E1 -2148.746,E2 -2148.746} C_VEL
LIN {X 0,Y 573.284,Z 169.889,A -85,B 0,C 180,E1 -2151.541,E2 -2151.541} C_VEL
LIN {X 0,Y 573.29,Z 169.891,A -85,B 0,C 180,E1 -2154.372,E2 -2154.372} C_VEL
LIN {X 0,Y 573.311,Z 169.888,A -85,B 0,C 180,E1 -2157.893,E2 -2157.893} C_VEL
LIN {X 0,Y 573.336,Z 169.881,A -85,B 0,C 180,E1 -2160.703,E2 -2160.703} C_VEL
LIN {X 0,Y 573.231,Z 169.896,A -85,B 0,C 180,E1 -2163.515,E2 -2163.515} C_VEL
LIN {X 0,Y 573.289,Z 169.888,A -85,B 0,C 180,E1 -2165.629,E2 -2165.629} C_VEL
LIN {X 0,Y 573.273,Z 169.889,A -85,B 0,C 180,E1 -2167.751,E2 -2167.751} C_VEL
LIN {X 0,Y 573.268,Z 169.893,A -85,B 0,C 180,E1 -2170.597,E2 -2170.597} C_VEL
LIN {X 0,Y 573.267,Z 169.893,A -85,B 0,C 180,E1 -2172.749,E2 -2172.749} C_VEL
LIN {X 0,Y 573.238,Z 169.895,A -85,B 0,C 180,E1 -2174.92,E2 -2174.92} C_VEL
LIN {X 0,Y 573.248,Z 169.893,A -85,B 0,C 180,E1 -2177.849,E2 -2177.849} C_VEL
LIN {X 0,Y 573.254,Z 169.892,A -85,B 0,C 180,E1 -2180.077,E2 -2180.077} C_VEL
LIN {X 0,Y 573.238,Z 169.897,A -85,B 0,C 180,E1 -2183.1,E2 -2183.1} C_VEL
LIN {X 0,Y 573.258,Z 169.894,A -85,B 0,C 180,E1 -2185.41,E2 -2185.41} C_VEL
LIN {X 0,Y 573.248,Z 169.893,A -85,B 0,C 180,E1 -2188.028,E2 -2188.028} C_VEL
LIN {X 0,Y 573.249,Z 169.894,A -85,B 0,C 180,E1 -2190.176,E2 -2190.176} C_VEL
LIN {X 0,Y 573.257,Z 169.892,A -85,B 0,C 180,E1 -2192.645,E2 -2192.645} C_VEL
LIN {X 0,Y 573.211,Z 169.897,A -85,B 0,C 180,E1 -2195.188,E2 -2195.188} C_VEL
LIN {X 0,Y 573.237,Z 169.895,A -85,B 0,C 180,E1 -2197.808,E2 -2197.808} C_VEL
LIN {X 0,Y 573.247,Z 169.894,A -85,B 0,C 180,E1 -2200.525,E2 -2200.525} C_VEL
LIN {X 0,Y 573.241,Z 169.894,A -85,B 0,C 180,E1 -2203.359,E2 -2203.359} C_VEL
LIN {X 0,Y 573.245,Z 169.894,A -85,B 0,C 180,E1 -2206.331,E2 -2206.331} C_VEL
LIN {X 0,Y 573.231,Z 169.896,A -85,B 0,C 180,E1 -2208.543,E2 -2208.543} C_VEL
LIN {X 0,Y 573.245,Z 169.893,A -85,B 0,C 180,E1 -2211.299,E2 -2211.299} C_VEL
LIN {X 0,Y 573.239,Z 169.898,A -85,B 0,C 180,E1 -2214.015,E2 -2214.015} C_VEL
LIN {X 0,Y 573.287,Z 169.892,A -85,B 0,C 180,E1 -2216.519,E2 -2216.519} C_VEL
LIN {X 0,Y 573.246,Z 169.932,A -85,B 0,C 180,E1 -2218.494,E2 -2218.494} C_VEL
LIN {X 0,Y 573.665,Z 172.995,A -85,B 0,C 180,E1 -2219.457,E2 -2219.457} C_VEL
LIN {X 0,Y 573.572,Z 181.158,A -85,B 0,C 180,E1 -2221.911,E2 -2221.911} C_VEL
LIN {X 0,Y 573.392,Z 190.429,A -85,B 0,C 180,E1 -2224.597,E2 -2224.597} C_VEL
LIN {X 0,Y 573.315,Z 198.915,A -85,B 0,C 180,E1 -2226.904,E2 -2226.904} C_VEL
LIN {X 0,Y 573.29,Z 208.788,A -85,B 0,C 180,E1 -2229.55,E2 -2229.55} C_VEL
LIN {X 0,Y 573.23,Z 219.845,A -85,B 0,C 180,E1 -2232.52,E2 -2232.52} C_VEL
LIN {X 0,Y 573.141,Z 230.794,A -85,B 0,C 180,E1 -2235.411,E2 -2235.411} C_VEL
LIN {X 0,Y 573.111,Z 241.969,A -85,B 0,C 180,E1 -2238.326,E2 -2238.326} C_VEL
LIN {X 0,Y 573.089,Z 249.091,A -85,B 0,C 180,E1 -2240.125,E2 -2240.125} C_VEL
LIN {X 0,Y 573.51,Z 255.585,A -85,B 0,C 180,E1 -2240.277,E2 -2240.277} C_VEL
LIN {X 0,Y 573.47,Z 264.892,A -85,B 0,C 180,E1 -2240.566,E2 -2240.566} C_VEL
LIN {X 0,Y 573.377,Z 273.399,A -85,B 0,C 180,E1 -2240.92,E2 -2240.92} C_VEL
LIN {X 0,Y 573.319,Z 281.731,A -85,B 0,C 180,E1 -2241.364,E2 -2241.364} C_VEL
LIN {X 0,Y 573.27,Z 289.771,A -85,B 0,C 180,E1 -2241.895,E2 -2241.895} C_VEL
LIN {X 0,Y 573.194,Z 298.432,A -85,B 0,C 180,E1 -2242.603,E2 -2242.603} C_VEL
LIN {X 0,Y 573.131,Z 306.472,A -85,B 0,C 180,E1 -2243.429,E2 -2243.429} C_VEL
LIN {X 0,Y 573.113,Z 312.435,A -85,B 0,C 180,E1 -2244.194,E2 -2244.194} C_VEL
LIN {X 0,Y 572.995,Z 317.989,A -85,B 0,C 180,E1 -2245.075,E2 -2245.075} C_VEL
LIN {X 0,Y 573.024,Z 323.149,A -85,B 0,C 180,E1 -2246.132,E2 -2246.132} C_VEL
LIN {X 0,Y 572.99,Z 325.789,A -85,B 0,C 180,E1 -2246.836,E2 -2246.836} C_VEL
LIN {X 0,Y 572.94,Z 328.682,A -85,B 0,C 180,E1 -2247.891,E2 -2247.891} C_VEL
LIN {X 0,Y 572.944,Z 329.935,A -85,B 0,C 180,E1 -2248.594,E2 -2248.594} C_VEL
LIN {X 0,Y 572.937,Z 330.71,A -85,B 0,C 180,E1 -2249.297,E2 -2249.297} C_VEL
LIN {X 0,Y 572.935,Z 331,A -85,B 0,C 180,E1 -2250,E2 -2250} C_VEL
LIN {X 0,Y 572.937,Z 330.709,A -85,B 0,C 180,E1 -2250.703,E2 -2250.703} C_VEL
LIN {X 0,Y 572.944,Z 329.934,A -85,B 0,C 180,E1 -2251.406,E2 -2251.406} C_VEL
LIN {X 0,Y 572.94,Z 328.681,A -85,B 0,C 180,E1 -2252.109,E2 -2252.109} C_VEL
LIN {X 0,Y 572.99,Z 325.787,A -85,B 0,C 180,E1 -2253.164,E2 -2253.164} C_VEL
LIN {X 0,Y 573.024,Z 323.147,A -85,B 0,C 180,E1 -2253.868,E2 -2253.868} C_VEL
LIN {X 0,Y 572.995,Z 317.985,A -85,B 0,C 180,E1 -2254.925,E2 -2254.925} C_VEL
LIN {X 0,Y 573.138,Z 311.185,A -85,B 0,C 180,E1 -2255.983,E2 -2255.983} C_VEL
LIN {X 0,Y 573.164,Z 303.803,A -85,B 0,C 180,E1 -2256.86,E2 -2256.86} C_VEL
LIN {X 0,Y 573.217,Z 296.403,A -85,B 0,C 180,E1 -2257.574,E2 -2257.574} C_VEL
LIN {X 0,Y 573.296,Z 288.541,A -85,B 0,C 180,E1 -2258.193,E2 -2258.193} C_VEL
LIN {X 0,Y 573.382,Z 278.726,A -85,B 0,C 180,E1 -2258.813,E2 -2258.813} C_VEL
LIN {X 0,Y 573.434,Z 267.299,A -85,B 0,C 180,E1 -2259.346,E2 -2259.346} C_VEL
LIN {X 0,Y 573.526,Z 257.24,A -85,B 0,C 180,E1 -2259.678,E2 -2259.678} C_VEL
LIN {X 0,Y 573.227,Z 250.377,A -85,B 0,C 180,E1 -2259.85,E2 -2259.85} C_VEL
LIN {X 0,Y 573.052,Z 248.882,A -85,B 0,C 180,E1 -2259.887,E2 -2259.887} C_VEL
LIN {X 0,Y 573.091,Z 239.203,A -85,B 0,C 180,E1 -2262.393,E2 -2262.393} C_VEL
LIN {X 0,Y 573.162,Z 228.141,A -85,B 0,C 180,E1 -2265.286,E2 -2265.286} C_VEL
LIN {X 0,Y 573.228,Z 217.079,A -85,B 0,C 180,E1 -2268.219,E2 -2268.219} C_VEL
LIN {X 0,Y 573.303,Z 207.285,A -85,B 0,C 180,E1 -2270.825,E2 -2270.825} C_VEL
LIN {X 0,Y 573.369,Z 195.994,A -85,B 0,C 180,E1 -2273.86,E2 -2273.86} C_VEL
LIN {X 0,Y 573.454,Z 186.492,A -85,B 0,C 180,E1 -2276.536,E2 -2276.536} C_VEL
LIN {X 0,Y 573.626,Z 176.942,A -85,B 0,C 180,E1 -2279.346,E2 -2279.346} C_VEL
LIN {X 0,Y 573.542,Z 171.525,A -85,B 0,C 180,E1 -2280.975,E2 -2280.975} C_VEL
LIN {X 0,Y 573.239,Z 169.897,A -85,B 0,C 180,E1 -2281.506,E2 -2281.506} C_VEL
LIN {X 0,Y 573.269,Z 169.891,A -85,B 0,C 180,E1 -2284.329,E2 -2284.329} C_VEL
LIN {X 0,Y 573.255,Z 169.891,A -85,B 0,C 180,E1 -2287.166,E2 -2287.166} C_VEL
LIN {X 0,Y 573.242,Z 169.892,A -85,B 0,C 180,E1 -2289.608,E2 -2289.608} C_VEL
LIN {X 0,Y 573.24,Z 169.894,A -85,B 0,C 180,E1 -2292.641,E2 -2292.641} C_VEL
LIN {X 0,Y 573.228,Z 169.897,A -85,B 0,C 180,E1 -2295.666,E2 -2295.666} C_VEL
LIN {X 0,Y 573.23,Z 169.894,A -85,B 0,C 180,E1 -2298.543,E2 -2298.543} C_VEL
LIN {X 0,Y 573.24,Z 169.892,A -85,B 0,C 180,E1 -2301.298,E2 -2301.298} C_VEL
LIN {X 0,Y 573.215,Z 169.896,A -85,B 0,C 180,E1 -2304.019,E2 -2304.019} C_VEL
LIN {X 0,Y 573.274,Z 169.889,A -85,B 0,C 180,E1 -2306.518,E2 -2306.518} C_VEL
LIN {X 0,Y 573.23,Z 169.894,A -85,B 0,C 180,E1 -2309.118,E2 -2309.118} C_VEL
LIN {X 0,Y 573.234,Z 169.893,A -85,B 0,C 180,E1 -2311.435,E2 -2311.435} C_VEL
LIN {X 0,Y 573.259,Z 169.894,A -85,B 0,C 180,E1 -2314.59,E2 -2314.59} C_VEL
LIN {X 0,Y 573.239,Z 169.893,A -85,B 0,C 180,E1 -2317.662,E2 -2317.662} C_VEL
LIN {X 0,Y 573.271,Z 169.889,A -85,B 0,C 180,E1 -2320.67,E2 -2320.67} C_VEL
LIN {X 0,Y 573.25,Z 169.895,A -85,B 0,C 180,E1 -2323.621,E2 -2323.621} C_VEL
LIN {X 0,Y 573.277,Z 169.889,A -85,B 0,C 180,E1 -2325.807,E2 -2325.807} C_VEL
LIN {X 0,Y 573.268,Z 169.893,A -85,B 0,C 180,E1 -2328.745,E2 -2328.745} C_VEL
LIN {X 0,Y 573.259,Z 169.892,A -85,B 0,C 180,E1 -2331.54,E2 -2331.54} C_VEL
LIN {X 0,Y 573.239,Z 169.896,A -85,B 0,C 180,E1 -2333.664,E2 -2333.664} C_VEL
LIN {X 0,Y 573.231,Z 169.894,A -85,B 0,C 180,E1 -2335.781,E2 -2335.781} C_VEL
LIN {X 0,Y 573.3,Z 169.886,A -85,B 0,C 180,E1 -2337.892,E2 -2337.892} C_VEL
